	(* After writting, it is necessary to check if the parameter has been writting correctly*)
	Voltage_Guard_Min_Error_L1_RD(
		sNetId:= netID_internal,
		nSlaveAddr := Slave_Add_global_assign, 
		nIndex:= 16#8001, 
		nSubIndex := 16#11, 
		pDstBuf:= ADR(Voltage_Guard_Min_Error_L1), 
		cbBufLen:=SIZEOF(Voltage_Guard_Min_Error_L1),
		bExecute:= Exec_READ_Voltage_Guard_Min_Error_L1);
	
	(* Logic to handle the errors in the reading*)	
	IF NOT Voltage_Guard_Min_Error_L1_RD.bBusy AND NOT Voltage_Guard_Min_Error_L1_WR.bBusy THEN
    	Exec_READ_Voltage_Guard_Min_Error_L1 := FALSE;
		IF NOT Voltage_Guard_Min_Error_L1_RD.bError THEN 
			(* write successful *)
			Error_Voltage_Guard_Min_Error_L1 := FALSE;
			Previous_Voltage_Guard_Min_Error_L1_val := Voltage_Guard_Min_Error_L1;
		ELSE 
			(* write failed *)
			Error_Voltage_Guard_Min_Error_L1 := Voltage_Guard_Min_Error_L1_RD.bError;
    END_IF

    Voltage_Guard_Min_Error_L1_RD(bExecute := FALSE);
	
	END_IF
(******************************** VOLTAGE GUARD MIN ERROR L1 *****************************************)

(********************************* VOLTAGE GUARD MIN ERROR L2 ****************************************)
	(* Execution of the writing reading of Voltage Guard Min Error L2. When the previous value is diferent to the
	current one, the is executed the command*)
	IF Voltage_Guard_Min_Error_L2 <> Previous_Voltage_Guard_Min_Error_L2_val THEN
		Exec_Voltage_Guard_Min_Error_L2 := TRUE;
	END_IF
	
	(* Function to write the new value in the CoE parameter*)
	Voltage_Guard_Min_Error_L2_WR(
		sNetId:= netID_internal, 
		nSlaveAddr:= Slave_Add_global_assign, 
		nSubIndex:= 16#11, 
		nIndex:= 16#8011, 
		pSrcBuf:= ADR(Voltage_Guard_Min_Error_L2), 
		cbBufLen:= SIZEOF(Voltage_Guard_Min_Error_L2), 
		bExecute:= Exec_Voltage_Guard_Min_Error_L2, 
		tTimeout:= T#1S);
	
	(* Logic to handle the errors and launch the reading*)	
	IF NOT Voltage_Guard_Min_Error_L2_WR.bBusy THEN
    	Exec_Voltage_Guard_Min_Error_L2 := FALSE;
		IF NOT Voltage_Guard_Min_Error_L2_WR.bError THEN 
			(* write successful *)
			Error_Voltage_Guard_Min_Error_L2 := FALSE;
			IF Previous_Voltage_Guard_Min_Error_L2_val <> Voltage_Guard_Min_Error_L2 THEN
				Previous_Voltage_Guard_Min_Error_L2_val := Voltage_Guard_Min_Error_L2;
				Exec_READ_Voltage_Guard_Min_Error_L2 := TRUE;
			END_IF
		ELSE 
			(* write failed *)
			Error_Voltage_Guard_Min_Error_L2 := Voltage_Guard_Min_Error_L2_WR.bError;
			Voltage_Guard_Min_Error_L2 := Previous_Voltage_Guard_Min_Error_L2_val;
		END_IF
	
		Voltage_Guard_Min_Error_L2_WR(bExecute := FALSE);
	
	END_IF
	
	(* After writting, it is necessary to check if the parameter has been writting correctly*)
	Voltage_Guard_Min_Error_L2_RD(
		sNetId:= netID_internal,
		nSlaveAddr := Slave_Add_global_assign, 
		nIndex:= 16#8011, 
		nSubIndex := 16#11, 
		pDstBuf:= ADR(Voltage_Guard_Min_Error_L2), 
		cbBufLen:=SIZEOF(Voltage_Guard_Min_Error_L2),
		bExecute:= Exec_READ_Voltage_Guard_Min_Error_L2);
	
	(* Logic to handle the errors in the reading*)	
	IF NOT Voltage_Guard_Min_Error_L2_RD.bBusy AND NOT Voltage_Guard_Min_Error_L2_WR.bBusy THEN
    	Exec_READ_Voltage_Guard_Min_Error_L2 := FALSE;
		IF NOT Voltage_Guard_Min_Error_L2_RD.bError THEN 
			(* write successful *)
			Error_Voltage_Guard_Min_Error_L2 := FALSE;
			Previous_Voltage_Guard_Min_Error_L2_val := Voltage_Guard_Min_Error_L2;
		ELSE 
			(* write failed *)
			Error_Voltage_Guard_Min_Error_L2 := Voltage_Guard_Min_Error_L2_RD.bError;
    END_IF

    Voltage_Guard_Min_Error_L2_RD(bExecute := FALSE);
	
	END_IF
(********************************* VOLTAGE GUARD MIN ERROR L2 ****************************************)

(********************************* VOLTAGE GUARD MIN ERROR L3 ****************************************)
	(* Execution of the writing reading of Voltage Guard Min Error L23. When the previous value is diferent to the
	current one, the is executed the command*)
	IF Voltage_Guard_Min_Error_L3 <> Previous_Voltage_Guard_Min_Error_L3_val THEN
		Exec_Voltage_Guard_Min_Error_L3 := TRUE;
	END_IF
	
	(* Function to write the new value in the CoE parameter*)
	Voltage_Guard_Min_Error_L3_WR(
		sNetId:= netID_internal, 
		nSlaveAddr:= Slave_Add_global_assign, 
		nSubIndex:= 16#11, 
		nIndex:= 16#8021, 
		pSrcBuf:= ADR(Voltage_Guard_Min_Error_L3), 
		cbBufLen:= SIZEOF(Voltage_Guard_Min_Error_L3), 
		bExecute:= Exec_Voltage_Guard_Min_Error_L3, 
		tTimeout:= T#1S);
	
	(* Logic to handle the errors and launch the reading*)	
	IF NOT Voltage_Guard_Min_Error_L3_WR.bBusy THEN
    	Exec_Voltage_Guard_Min_Error_L3 := FALSE;
		IF NOT Voltage_Guard_Min_Error_L3_WR.bError THEN 
			(* write successful *)
			Error_Voltage_Guard_Min_Error_L3 := FALSE;
			IF Previous_Voltage_Guard_Min_Error_L3_val <> Voltage_Guard_Min_Error_L3 THEN
				Previous_Voltage_Guard_Min_Error_L3_val := Voltage_Guard_Min_Error_L3;
				Exec_READ_Voltage_Guard_Min_Error_L3 := TRUE;
			END_IF
		ELSE 
			(* write failed *)
			Error_Voltage_Guard_Min_Error_L3 := Voltage_Guard_Min_Error_L3_WR.bError;
			Voltage_Guard_Min_Error_L3 := Previous_Voltage_Guard_Min_Error_L3_val;
		END_IF
	
		Voltage_Guard_Min_Error_L3_WR(bExecute := FALSE);
	
	END_IF
	
	(* After writting, it is necessary to check if the parameter has been writting correctly*)
	Voltage_Guard_Min_Error_L3_RD(
		sNetId:= netID_internal,
		nSlaveAddr := Slave_Add_global_assign, 
		nIndex:= 16#8021, 
		nSubIndex := 16#11, 
		pDstBuf:= ADR(Voltage_Guard_Min_Error_L3), 
		cbBufLen:=SIZEOF(Voltage_Guard_Min_Error_L3),
		bExecute:= Exec_READ_Voltage_Guard_Min_Error_L3);
	
	(* Logic to handle the errors in the reading*)	
	IF NOT Voltage_Guard_Min_Error_L3_RD.bBusy AND NOT Voltage_Guard_Min_Error_L3_WR.bBusy THEN
    	Exec_READ_Voltage_Guard_Min_Error_L3 := FALSE;
		IF NOT Voltage_Guard_Min_Error_L3_RD.bError THEN 
			(* write successful *)
			Error_Voltage_Guard_Min_Error_L3 := FALSE;
			Previous_Voltage_Guard_Min_Error_L3_val := Voltage_Guard_Min_Error_L3;
		ELSE 
			(* write failed *)
			Error_Voltage_Guard_Min_Error_L3 := Voltage_Guard_Min_Error_L3_RD.bError;
    END_IF

    Voltage_Guard_Min_Error_L3_RD(bExecute := FALSE);
	
	END_IF
(******************************** VOLTAGE GUARD MIN ERROR L3 *****************************************)

(********************************* VOLTAGE GUARD MIN WARNING L1 **************************************)
	(* Execution of the writing reading of Voltage Guard Min Error L1. When the previous value is diferent to the
	current one, the is executed the command*)
	IF Voltage_Guard_Min_Warning_L1 <> Previous_Voltage_Guard_Min_Warning_L1_val THEN
		Exec_Voltage_Guard_Min_Warning_L1 := TRUE;
	END_IF
	
	(* Function to write the new value in the CoE parameter*)
	Voltage_Guard_Min_Warning_L1_WR(
		sNetId:= netID_internal, 
		nSlaveAddr:= Slave_Add_global_assign, 
		nSubIndex:= 16#12, 
		nIndex:= 16#8001, 
		pSrcBuf:= ADR(Voltage_Guard_Min_Warning_L1), 
		cbBufLen:= SIZEOF(Voltage_Guard_Min_Warning_L1), 
		bExecute:= Exec_Voltage_Guard_Min_Warning_L1, 
		tTimeout:= T#1S);
	
	(* Logic to handle the errors and launch the reading*)	
	IF NOT Voltage_Guard_Min_Warning_L1_WR.bBusy THEN
    	Exec_Voltage_Guard_Min_Warning_L1 := FALSE;
		IF NOT Voltage_Guard_Min_Warning_L1_WR.bError THEN 
			(* write successful *)
			Error_Voltage_Guard_Min_Warning_L1 := FALSE;
			IF Previous_Voltage_Guard_Min_Warning_L1_val <> Voltage_Guard_Min_Warning_L1 THEN
				Previous_Voltage_Guard_Min_Warning_L1_val := Voltage_Guard_Min_Warning_L1;
				Exec_READ_Voltage_Guard_Min_Warning_L1 := TRUE;
			END_IF
		ELSE 
			(* write failed *)
			Error_Voltage_Guard_Min_Warning_L1 := Voltage_Guard_Min_Warning_L1_WR.bError;
			Voltage_Guard_Min_Warning_L1 := Previous_Voltage_Guard_Min_Warning_L1_val;
		END_IF
	
		Voltage_Guard_Min_Warning_L1_WR(bExecute := FALSE);
	
	END_IF
	
	(* After writting, it is necessary to check if the parameter has been writting correctly*)
	Voltage_Guard_Min_Warning_L1_RD(
		sNetId:= netID_internal,
		nSlaveAddr := Slave_Add_global_assign, 
		nIndex:= 16#8001, 
		nSubIndex := 16#12, 
		pDstBuf:= ADR(Voltage_Guard_Min_Warning_L1), 
		cbBufLen:=SIZEOF(Voltage_Guard_Min_Warning_L1),
		bExecute:= Exec_READ_Voltage_Guard_Min_Warning_L1);
	
	(* Logic to handle the errors in the reading*)	
	IF NOT Voltage_Guard_Min_Warning_L1_RD.bBusy AND NOT Voltage_Guard_Min_Warning_L1_WR.bBusy THEN
    	Exec_READ_Voltage_Guard_Min_Warning_L1 := FALSE;
		IF NOT Voltage_Guard_Min_Warning_L1_RD.bError THEN 
			(* write successful *)
			Error_Voltage_Guard_Min_Warning_L1 := FALSE;
			Previous_Voltage_Guard_Min_Warning_L1_val := Voltage_Guard_Min_Warning_L1;
		ELSE 
			(* write failed *)
			Error_Voltage_Guard_Min_Warning_L1 := Voltage_Guard_Min_Warning_L1_RD.bError;
    END_IF

    Voltage_Guard_Min_Warning_L1_RD(bExecute := FALSE);
	
	END_IF
(********************************* VOLTAGE GUARD MIN WARNING L1 **************************************)

(********************************* VOLTAGE GUARD MIN WARNING L2 **************************************)
	(* Execution of the writing reading of Voltage Guard Min Error L2. When the previous value is diferent to the
	current one, the is executed the command*)
	IF Voltage_Guard_Min_Warning_L2 <> Previous_Voltage_Guard_Min_Warning_L2_val THEN
		Exec_Voltage_Guard_Min_Warning_L2 := TRUE;
	END_IF
	
	(* Function to write the new value in the CoE parameter*)
	Voltage_Guard_Min_Warning_L2_WR(
		sNetId:= netID_internal, 
		nSlaveAddr:= Slave_Add_global_assign, 
		nSubIndex:= 16#12, 
		nIndex:= 16#8011, 
		pSrcBuf:= ADR(Voltage_Guard_Min_Warning_L2), 
		cbBufLen:= SIZEOF(Voltage_Guard_Min_Warning_L2), 
		bExecute:= Exec_Voltage_Guard_Min_Warning_L2, 
		tTimeout:= T#1S);
	
	(* Logic to handle the errors and launch the reading*)	
	IF NOT Voltage_Guard_Min_Warning_L2_WR.bBusy THEN
    	Exec_Voltage_Guard_Min_Warning_L2 := FALSE;
		IF NOT Voltage_Guard_Min_Warning_L2_WR.bError THEN 
			(* write successful *)
			Error_Voltage_Guard_Min_Warning_L2 := FALSE;
			IF Previous_Voltage_Guard_Min_Warning_L2_val <> Voltage_Guard_Min_Warning_L2 THEN
				Previous_Voltage_Guard_Min_Warning_L2_val := Voltage_Guard_Min_Warning_L2;
				Exec_READ_Voltage_Guard_Min_Warning_L2 := TRUE;
			END_IF
		ELSE 
			(* write failed *)
			Error_Voltage_Guard_Min_Warning_L2 := Voltage_Guard_Min_Warning_L2_WR.bError;
			Voltage_Guard_Min_Warning_L2 := Previous_Voltage_Guard_Min_Warning_L2_val;
		END_IF
	
		Voltage_Guard_Min_Warning_L2_WR(bExecute := FALSE);
	
	END_IF
	
	(* After writting, it is necessary to check if the parameter has been writting correctly*)
	Voltage_Guard_Min_Warning_L2_RD(
		sNetId:= netID_internal,
		nSlaveAddr := Slave_Add_global_assign, 
		nIndex:= 16#8011, 
		nSubIndex := 16#12, 
		pDstBuf:= ADR(Voltage_Guard_Min_Warning_L2), 
		cbBufLen:=SIZEOF(Voltage_Guard_Min_Warning_L2),
		bExecute:= Exec_READ_Voltage_Guard_Min_Warning_L2);
	
	(* Logic to handle the errors in the reading*)	
	IF NOT Voltage_Guard_Min_Warning_L2_RD.bBusy AND NOT Voltage_Guard_Min_Warning_L2_WR.bBusy THEN
    	Exec_READ_Voltage_Guard_Min_Warning_L2 := FALSE;
		IF NOT Voltage_Guard_Min_Warning_L2_RD.bError THEN 
			(* write successful *)
			Error_Voltage_Guard_Min_Warning_L2 := FALSE;
			Previous_Voltage_Guard_Min_Warning_L2_val := Voltage_Guard_Min_Warning_L2;
		ELSE 
			(* write failed *)
			Error_Voltage_Guard_Min_Warning_L2 := Voltage_Guard_Min_Warning_L2_RD.bError;
    END_IF

    Voltage_Guard_Min_Warning_L2_RD(bExecute := FALSE);
	
	END_IF
(********************************* VOLTAGE GUARD MIN WARNING L2 ***************************************)

(********************************* VOLTAGE GUARD MIN WARNING L3 **************************************)
	(* Execution of the writing reading of Voltage Guard Min Error L3. When the previous value is diferent to the
	current one, the is executed the command*)
	IF Voltage_Guard_Min_Warning_L3 <> Previous_Voltage_Guard_Min_Warning_L3_val THEN
		Exec_Voltage_Guard_Min_Warning_L3 := TRUE;
	END_IF
	
	(* Function to write the new value in the CoE parameter*)
	Voltage_Guard_Min_Warning_L3_WR(
		sNetId:= netID_internal, 
		nSlaveAddr:= Slave_Add_global_assign, 
		nSubIndex:= 16#12, 
		nIndex:= 16#8021, 
		pSrcBuf:= ADR(Voltage_Guard_Min_Warning_L3), 
		cbBufLen:= SIZEOF(Voltage_Guard_Min_Warning_L3), 
		bExecute:= Exec_Voltage_Guard_Min_Warning_L3, 
		tTimeout:= T#1S);
	
	(* Logic to handle the errors and launch the reading*)	
	IF NOT Voltage_Guard_Min_Warning_L3_WR.bBusy THEN
    	Exec_Voltage_Guard_Min_Warning_L3 := FALSE;
		IF NOT Voltage_Guard_Min_Warning_L3_WR.bError THEN 
			(* write successful *)
			Error_Voltage_Guard_Min_Warning_L3 := FALSE;
			IF Previous_Voltage_Guard_Min_Warning_L3_val <> Voltage_Guard_Min_Warning_L3 THEN
				Previous_Voltage_Guard_Min_Warning_L3_val := Voltage_Guard_Min_Warning_L3;
				Exec_READ_Voltage_Guard_Min_Warning_L3 := TRUE;
			END_IF
		ELSE 
			(* write failed *)
			Error_Voltage_Guard_Min_Warning_L3 := Voltage_Guard_Min_Warning_L3_WR.bError;
			Voltage_Guard_Min_Warning_L3 := Previous_Voltage_Guard_Min_Warning_L3_val;
		END_IF
	
		Voltage_Guard_Min_Warning_L3_WR(bExecute := FALSE);
	
	END_IF
	
	(* After writting, it is necessary to check if the parameter has been writting correctly*)
	Voltage_Guard_Min_Warning_L3_RD(
		sNetId:= netID_internal,
		nSlaveAddr := Slave_Add_global_assign, 
		nIndex:= 16#8021, 
		nSubIndex := 16#12, 
		pDstBuf:= ADR(Voltage_Guard_Min_Warning_L3), 
		cbBufLen:=SIZEOF(Voltage_Guard_Min_Warning_L3),
		bExecute:= Exec_READ_Voltage_Guard_Min_Warning_L3);
	
	(* Logic to handle the errors in the reading*)	
	IF NOT Voltage_Guard_Min_Warning_L3_RD.bBusy AND NOT Voltage_Guard_Min_Warning_L3_WR.bBusy THEN
    	Exec_READ_Voltage_Guard_Min_Warning_L3 := FALSE;
		IF NOT Voltage_Guard_Min_Warning_L3_RD.bError THEN 
			(* write successful *)
			Error_Voltage_Guard_Min_Warning_L3 := FALSE;
			Previous_Voltage_Guard_Min_Warning_L3_val := Voltage_Guard_Min_Warning_L3;
		ELSE 
			(* write failed *)
			Error_Voltage_Guard_Min_Warning_L3 := Voltage_Guard_Min_Warning_L3_RD.bError;
    END_IF

    Voltage_Guard_Min_Warning_L3_RD(bExecute := FALSE);
	
	END_IF
(********************************* VOLTAGE GUARD MIN WARNING L3 ***************************************)

(********************************* VOLTAGE GUARD MAX WARNING L1 **************************************)
	(* Execution of the writing reading of Voltage Guard Max Warning L1. When the previous value is diferent to the
	current one, the is executed the command*)
	IF Voltage_Guard_Max_Warning_L1 <> Previous_Voltage_Guard_Max_Warning_L1_val THEN
		Exec_Voltage_Guard_Max_Warning_L1 := TRUE;
	END_IF
	
	(* Function to write the new value in the CoE parameter*)
	Voltage_Guard_Max_Warning_L1_WR(
		sNetId:= netID_internal, 
		nSlaveAddr:= Slave_Add_global_assign, 
		nSubIndex:= 16#13, 
		nIndex:= 16#8001, 
		pSrcBuf:= ADR(Voltage_Guard_Max_Warning_L1), 
		cbBufLen:= SIZEOF(Voltage_Guard_Max_Warning_L1), 
		bExecute:= Exec_Voltage_Guard_Max_Warning_L1, 
		tTimeout:= T#1S);
	
	(* Logic to handle the errors and launch the reading*)	
	IF NOT Voltage_Guard_Max_Warning_L1_WR.bBusy THEN
    	Exec_Voltage_Guard_Max_Warning_L1 := FALSE;
		IF NOT Voltage_Guard_Max_Warning_L1_WR.bError THEN 
			(* write successful *)
			Error_Voltage_Guard_Max_Warning_L1 := FALSE;
			IF Previous_Voltage_Guard_Max_Warning_L1_val <> Voltage_Guard_Max_Warning_L1 THEN
				Previous_Voltage_Guard_Max_Warning_L1_val := Voltage_Guard_Max_Warning_L1;
				Exec_READ_Voltage_Guard_Max_Warning_L1 := TRUE;
			END_IF
		ELSE 
			(* write failed *)
			Error_Voltage_Guard_Max_Warning_L1 := Voltage_Guard_Max_Warning_L1_WR.bError;
			Voltage_Guard_Max_Warning_L1 := Previous_Voltage_Guard_Max_Warning_L1_val;
		END_IF
	
		Voltage_Guard_Max_Warning_L1_WR(bExecute := FALSE);
	
	END_IF
	
	(* After writting, it is necessary to check if the parameter has been writting correctly*)
	Voltage_Guard_Max_Warning_L1_RD(
		sNetId:= netID_internal,
		nSlaveAddr := Slave_Add_global_assign, 
		nIndex:= 16#8001, 
		nSubIndex := 16#13, 
		pDstBuf:= ADR(Voltage_Guard_Max_Warning_L1), 
		cbBufLen:=SIZEOF(Voltage_Guard_Max_Warning_L1),
		bExecute:= Exec_READ_Voltage_Guard_Max_Warning_L1);
	
	(* Logic to handle the errors in the reading*)	
	IF NOT Voltage_Guard_Max_Warning_L1_RD.bBusy AND NOT Voltage_Guard_Max_Warning_L1_WR.bBusy THEN
    	Exec_READ_Voltage_Guard_Max_Warning_L1 := FALSE;
		IF NOT Voltage_Guard_Max_Warning_L1_RD.bError THEN 
			(* write successful *)
			Error_Voltage_Guard_Max_Warning_L1 := FALSE;
			Previous_Voltage_Guard_Max_Warning_L1_val := Voltage_Guard_Max_Warning_L1;
		ELSE 
			(* write failed *)
			Error_Voltage_Guard_Max_Warning_L1 := Voltage_Guard_Max_Warning_L1_RD.bError;
    END_IF

    Voltage_Guard_Max_Warning_L1_RD(bExecute := FALSE);
	
	END_IF
(********************************* VOLTAGE GUARD MAX WARNING L1 **************************************)

(********************************* VOLTAGE GUARD MAX WARNING L2 **************************************)
	(* Execution of the writing reading of Voltage Guard Max Warning L2. When the previous value is diferent to the
	current one, the is executed the command*)
	IF Voltage_Guard_Max_Warning_L2 <> Previous_Voltage_Guard_Max_Warning_L2_val THEN
		Exec_Voltage_Guard_Max_Warning_L2 := TRUE;
	END_IF
	
	(* Function to write the new value in the CoE parameter*)
	Voltage_Guard_Max_Warning_L2_WR(
		sNetId:= netID_internal, 
		nSlaveAddr:= Slave_Add_global_assign, 
		nSubIndex:= 16#13, 
		nIndex:= 16#8011, 
		pSrcBuf:= ADR(Voltage_Guard_Max_Warning_L2), 
		cbBufLen:= SIZEOF(Voltage_Guard_Max_Warning_L2), 
		bExecute:= Exec_Voltage_Guard_Max_Warning_L2, 
		tTimeout:= T#1S);
	
	(* Logic to handle the errors and launch the reading*)	
	IF NOT Voltage_Guard_Max_Warning_L2_WR.bBusy THEN
    	Exec_Voltage_Guard_Max_Warning_L2 := FALSE;
		IF NOT Voltage_Guard_Max_Warning_L2_WR.bError THEN 
			(* write successful *)
			Error_Voltage_Guard_Max_Warning_L2 := FALSE;
			IF Previous_Voltage_Guard_Max_Warning_L2_val <> Voltage_Guard_Max_Warning_L2 THEN
				Previous_Voltage_Guard_Max_Warning_L2_val := Voltage_Guard_Max_Warning_L2;
				Exec_READ_Voltage_Guard_Max_Warning_L2 := TRUE;
			END_IF
		ELSE 
			(* write failed *)
			Error_Voltage_Guard_Max_Warning_L2 := Voltage_Guard_Max_Warning_L2_WR.bError;
			Voltage_Guard_Max_Warning_L2 := Previous_Voltage_Guard_Max_Warning_L2_val;
		END_IF
	
		Voltage_Guard_Max_Warning_L2_WR(bExecute := FALSE);
	
	END_IF
	
	(* After writting, it is necessary to check if the parameter has been writting correctly*)
	Voltage_Guard_Max_Warning_L2_RD(
		sNetId:= netID_internal,
		nSlaveAddr := Slave_Add_global_assign, 
		nIndex:= 16#8011, 
		nSubIndex := 16#13, 
		pDstBuf:= ADR(Voltage_Guard_Max_Warning_L2), 
		cbBufLen:=SIZEOF(Voltage_Guard_Max_Warning_L2),
		bExecute:= Exec_READ_Voltage_Guard_Max_Warning_L2);
	
	(* Logic to handle the errors in the reading*)	
	IF NOT Voltage_Guard_Max_Warning_L2_RD.bBusy AND NOT Voltage_Guard_Max_Warning_L2_WR.bBusy THEN
    	Exec_READ_Voltage_Guard_Max_Warning_L2 := FALSE;
		IF NOT Voltage_Guard_Max_Warning_L2_RD.bError THEN 
			(* write successful *)
			Error_Voltage_Guard_Max_Warning_L2 := FALSE;
			Previous_Voltage_Guard_Max_Warning_L2_val := Voltage_Guard_Max_Warning_L2;
		ELSE 
			(* write failed *)
			Error_Voltage_Guard_Max_Warning_L2 := Voltage_Guard_Max_Warning_L2_RD.bError;
    END_IF

    Voltage_Guard_Max_Warning_L2_RD(bExecute := FALSE);
	
	END_IF
(********************************* VOLTAGE GUARD MAX WARNING L2 **************************************)

(********************************* VOLTAGE GUARD MAX WARNING L3 **************************************)
	(* Execution of the writing reading of Voltage Guard Max Warning L3. When the previous value is diferent to the
	current one, the is executed the command*)
	IF Voltage_Guard_Max_Warning_L3 <> Previous_Voltage_Guard_Max_Warning_L3_val THEN
		Exec_Voltage_Guard_Max_Warning_L3 := TRUE;
	END_IF
	
	(* Function to write the new value in the CoE parameter*)
	Voltage_Guard_Max_Warning_L3_WR(
		sNetId:= netID_internal, 
		nSlaveAddr:= Slave_Add_global_assign, 
		nSubIndex:= 16#13, 
		nIndex:= 16#8021, 
		pSrcBuf:= ADR(Voltage_Guard_Max_Warning_L3), 
		cbBufLen:= SIZEOF(Voltage_Guard_Max_Warning_L3), 
		bExecute:= Exec_Voltage_Guard_Max_Warning_L3, 
		tTimeout:= T#1S);
	
	(* Logic to handle the errors and launch the reading*)	
	IF NOT Voltage_Guard_Max_Warning_L3_WR.bBusy THEN
    	Exec_Voltage_Guard_Max_Warning_L3 := FALSE;
		IF NOT Voltage_Guard_Max_Warning_L3_WR.bError THEN 
			(* write successful *)
			Error_Voltage_Guard_Max_Warning_L3 := FALSE;
			IF Previous_Voltage_Guard_Max_Warning_L3_val <> Voltage_Guard_Max_Warning_L3 THEN
				Previous_Voltage_Guard_Max_Warning_L3_val := Voltage_Guard_Max_Warning_L3;
				Exec_READ_Voltage_Guard_Max_Warning_L3 := TRUE;
			END_IF
		ELSE 
			(* write failed *)
			Error_Voltage_Guard_Max_Warning_L3 := Voltage_Guard_Max_Warning_L3_WR.bError;
			Voltage_Guard_Max_Warning_L3 := Previous_Voltage_Guard_Max_Warning_L3_val;
		END_IF
	
		Voltage_Guard_Max_Warning_L3_WR(bExecute := FALSE);
	
	END_IF
	
	(* After writting, it is necessary to check if the parameter has been writting correctly*)
	Voltage_Guard_Max_Warning_L3_RD(
		sNetId:= netID_internal,
		nSlaveAddr := Slave_Add_global_assign, 
		nIndex:= 16#8021, 
		nSubIndex := 16#13, 
		pDstBuf:= ADR(Voltage_Guard_Max_Warning_L3), 
		cbBufLen:=SIZEOF(Voltage_Guard_Max_Warning_L3),
		bExecute:= Exec_READ_Voltage_Guard_Max_Warning_L3);
	
	(* Logic to handle the errors in the reading*)	
	IF NOT Voltage_Guard_Max_Warning_L3_RD.bBusy AND NOT Voltage_Guard_Max_Warning_L3_WR.bBusy THEN
    	Exec_READ_Voltage_Guard_Max_Warning_L3 := FALSE;
		IF NOT Voltage_Guard_Max_Warning_L3_RD.bError THEN 
			(* write successful *)
			Error_Voltage_Guard_Max_Warning_L3 := FALSE;
			Previous_Voltage_Guard_Max_Warning_L3_val := Voltage_Guard_Max_Warning_L3;
		ELSE 
			(* write failed *)
			Error_Voltage_Guard_Max_Warning_L3 := Voltage_Guard_Max_Warning_L3_RD.bError;
    END_IF

    Voltage_Guard_Max_Warning_L3_RD(bExecute := FALSE);
	
	END_IF
(********************************* VOLTAGE GUARD MAX WARNING L3 **************************************)

(********************************* VOLTAGE GUARD MAX ERROR L1 ****************************************)
	(* Execution of the writing reading of Voltage Guard Max Error L1. When the previous value is diferent to the
	current one, the is executed the command*)
	IF Voltage_Guard_Max_Error_L1 <> Previous_Voltage_Guard_Max_Error_L1_val THEN
		Exec_Voltage_Guard_Max_Error_L1 := TRUE;
	END_IF
	
	(* Function to write the new value in the CoE parameter*)
	Voltage_Guard_Max_Error_L1_WR(
		sNetId:= netID_internal, 
		nSlaveAddr:= Slave_Add_global_assign, 
		nSubIndex:= 16#14, 
		nIndex:= 16#8001, 
		pSrcBuf:= ADR(Voltage_Guard_Max_Error_L1), 
		cbBufLen:= SIZEOF(Voltage_Guard_Max_Error_L1), 
		bExecute:= Exec_Voltage_Guard_Max_Error_L1, 
		tTimeout:= T#1S);
	
	(* Logic to handle the errors and launch the reading*)	
	IF NOT Voltage_Guard_Max_Error_L1_WR.bBusy THEN
    	Exec_Voltage_Guard_Max_Error_L1 := FALSE;
		IF NOT Voltage_Guard_Max_Error_L1_WR.bError THEN 
			(* write successful *)
			Error_Voltage_Guard_Max_Error_L1 := FALSE;
			IF Previous_Voltage_Guard_Max_Error_L1_val <> Voltage_Guard_Max_Error_L1 THEN
				Previous_Voltage_Guard_Max_Error_L1_val := Voltage_Guard_Max_Error_L1;
				Exec_READ_Voltage_Guard_Max_Error_L1 := TRUE;
			END_IF
		ELSE 
			(* write failed *)
			Error_Voltage_Guard_Max_Error_L1 := Voltage_Guard_Max_Error_L1_WR.bError;
			Voltage_Guard_Max_Error_L1 := Previous_Voltage_Guard_Max_Error_L1_val;
		END_IF
	
		Voltage_Guard_Max_Error_L1_WR(bExecute := FALSE);
	
	END_IF
	
	(* After writting, it is necessary to check if the parameter has been writting correctly*)
	Voltage_Guard_Max_Error_L1_RD(
		sNetId:= netID_internal,
		nSlaveAddr := Slave_Add_global_assign, 
		nIndex:= 16#8001, 
		nSubIndex := 16#14, 
		pDstBuf:= ADR(Voltage_Guard_Max_Error_L1), 
		cbBufLen:=SIZEOF(Voltage_Guard_Max_Error_L1),
		bExecute:= Exec_READ_Voltage_Guard_Max_Error_L1);
	
	(* Logic to handle the errors in the reading*)	
	IF NOT Voltage_Guard_Max_Error_L1_RD.bBusy AND NOT Voltage_Guard_Max_Error_L1_WR.bBusy THEN
    	Exec_READ_Voltage_Guard_Max_Error_L1 := FALSE;
		IF NOT Voltage_Guard_Max_Error_L1_RD.bError THEN 
			(* write successful *)
			Error_Voltage_Guard_Max_Error_L1 := FALSE;
			Previous_Voltage_Guard_Max_Error_L1_val := Voltage_Guard_Max_Error_L1;
		ELSE 
			(* write failed *)
			Error_Voltage_Guard_Max_Error_L1 := Voltage_Guard_Max_Error_L1_RD.bError;
    END_IF

    Voltage_Guard_Max_Error_L1_RD(bExecute := FALSE);
	
	END_IF
(******************************** VOLTAGE GUARD MAX ERROR L1 *****************************************)

(********************************* VOLTAGE GUARD MAX ERROR L2 ****************************************)
	(* Execution of the writing reading of Voltage Guard Max Error L2. When the previous value is diferent to the
	current one, the is executed the command*)
	IF Voltage_Guard_Max_Error_L2 <> Previous_Voltage_Guard_Max_Error_L2_val THEN
		Exec_Voltage_Guard_Max_Error_L2 := TRUE;
	END_IF
	
	(* Function to write the new value in the CoE parameter*)
	Voltage_Guard_Max_Error_L2_WR(
		sNetId:= netID_internal, 
		nSlaveAddr:= Slave_Add_global_assign, 
		nSubIndex:= 16#14, 
		nIndex:= 16#8011, 
		pSrcBuf:= ADR(Voltage_Guard_Max_Error_L2), 
		cbBufLen:= SIZEOF(Voltage_Guard_Max_Error_L2), 
		bExecute:= Exec_Voltage_Guard_Max_Error_L2, 
		tTimeout:= T#1S);
	
	(* Logic to handle the errors and launch the reading*)	
	IF NOT Voltage_Guard_Max_Error_L2_WR.bBusy THEN
    	Exec_Voltage_Guard_Max_Error_L2 := FALSE;
		IF NOT Voltage_Guard_Max_Error_L2_WR.bError THEN 
			(* write successful *)
			Error_Voltage_Guard_Max_Error_L2 := FALSE;
			IF Previous_Voltage_Guard_Max_Error_L2_val <> Voltage_Guard_Max_Error_L2 THEN
				Previous_Voltage_Guard_Max_Error_L2_val := Voltage_Guard_Max_Error_L2;
				Exec_READ_Voltage_Guard_Max_Error_L2 := TRUE;
			END_IF
		ELSE 
			(* write failed *)
			Error_Voltage_Guard_Max_Error_L2 := Voltage_Guard_Max_Error_L2_WR.bError;
			Voltage_Guard_Max_Error_L2 := Previous_Voltage_Guard_Max_Error_L2_val;
		END_IF
	
		Voltage_Guard_Max_Error_L2_WR(bExecute := FALSE);
	
	END_IF
	
	(* After writting, it is necessary to check if the parameter has been writting correctly*)
	Voltage_Guard_Max_Error_L2_RD(
		sNetId:= netID_internal,
		nSlaveAddr := Slave_Add_global_assign, 
		nIndex:= 16#8011, 
		nSubIndex := 16#14, 
		pDstBuf:= ADR(Voltage_Guard_Max_Error_L2), 
		cbBufLen:=SIZEOF(Voltage_Guard_Max_Error_L2),
		bExecute:= Exec_READ_Voltage_Guard_Max_Error_L2);
	
	(* Logic to handle the errors in the reading*)	
	IF NOT Voltage_Guard_Max_Error_L2_RD.bBusy AND NOT Voltage_Guard_Max_Error_L2_WR.bBusy THEN
    	Exec_READ_Voltage_Guard_Max_Error_L2 := FALSE;
		IF NOT Voltage_Guard_Max_Error_L2_RD.bError THEN 
			(* write successful *)
			Error_Voltage_Guard_Max_Error_L2 := FALSE;
			Previous_Voltage_Guard_Max_Error_L2_val := Voltage_Guard_Max_Error_L2;
		ELSE 
			(* write failed *)
			Error_Voltage_Guard_Max_Error_L2 := Voltage_Guard_Max_Error_L2_RD.bError;
    END_IF

    Voltage_Guard_Max_Error_L2_RD(bExecute := FALSE);
	
	END_IF
(******************************** VOLTAGE GUARD MAX ERROR L2 *****************************************)

(********************************* VOLTAGE GUARD MAX ERROR L3 ****************************************)
	(* Execution of the writing reading of Voltage Guard Max Error L3. When the previous value is diferent to the
	current one, the is executed the command*)
	IF Voltage_Guard_Max_Error_L3 <> Previous_Voltage_Guard_Max_Error_L3_val THEN
		Exec_Voltage_Guard_Max_Error_L3 := TRUE;
	END_IF
	
	(* Function to write the new value in the CoE parameter*)
	Voltage_Guard_Max_Error_L3_WR(
		sNetId:= netID_internal, 
		nSlaveAddr:= Slave_Add_global_assign, 
		nSubIndex:= 16#14, 
		nIndex:= 16#8021, 
		pSrcBuf:= ADR(Voltage_Guard_Max_Error_L3), 
		cbBufLen:= SIZEOF(Voltage_Guard_Max_Error_L3), 
		bExecute:= Exec_Voltage_Guard_Max_Error_L3, 
		tTimeout:= T#1S);
	
	(* Logic to handle the errors and launch the reading*)	
	IF NOT Voltage_Guard_Max_Error_L3_WR.bBusy THEN
    	Exec_Voltage_Guard_Max_Error_L3 := FALSE;
		IF NOT Voltage_Guard_Max_Error_L3_WR.bError THEN 
			(* write successful *)
			Error_Voltage_Guard_Max_Error_L3 := FALSE;
			IF Previous_Voltage_Guard_Max_Error_L3_val <> Voltage_Guard_Max_Error_L3 THEN
				Previous_Voltage_Guard_Max_Error_L3_val := Voltage_Guard_Max_Error_L3;
				Exec_READ_Voltage_Guard_Max_Error_L3 := TRUE;
			END_IF
		ELSE 
			(* write failed *)
			Error_Voltage_Guard_Max_Error_L3 := Voltage_Guard_Max_Error_L3_WR.bError;
			Voltage_Guard_Max_Error_L3 := Previous_Voltage_Guard_Max_Error_L3_val;
		END_IF
	
		Voltage_Guard_Max_Error_L3_WR(bExecute := FALSE);
	
	END_IF
	
	(* After writting, it is necessary to check if the parameter has been writting correctly*)
	Voltage_Guard_Max_Error_L3_RD(
		sNetId:= netID_internal,
		nSlaveAddr := Slave_Add_global_assign, 
		nIndex:= 16#8021, 
		nSubIndex := 16#14, 
		pDstBuf:= ADR(Voltage_Guard_Max_Error_L3), 
		cbBufLen:=SIZEOF(Voltage_Guard_Max_Error_L3),
		bExecute:= Exec_READ_Voltage_Guard_Max_Error_L3);
	
	(* Logic to handle the errors in the reading*)	
	IF NOT Voltage_Guard_Max_Error_L3_RD.bBusy AND NOT Voltage_Guard_Max_Error_L3_WR.bBusy THEN
    	Exec_READ_Voltage_Guard_Max_Error_L3 := FALSE;
		IF NOT Voltage_Guard_Max_Error_L3_RD.bError THEN 
			(* write successful *)
			Error_Voltage_Guard_Max_Error_L3 := FALSE;
			Previous_Voltage_Guard_Max_Error_L3_val := Voltage_Guard_Max_Error_L3;
		ELSE 
			(* write failed *)
			Error_Voltage_Guard_Max_Error_L3 := Voltage_Guard_Max_Error_L3_RD.bError;
    END_IF

    Voltage_Guard_Max_Error_L3_RD(bExecute := FALSE);
	
	END_IF
(******************************** VOLTAGE GUARD MAX ERROR L3 *****************************************)

END_IF

IF EL3_Selection = 'EL3453' THEN
	
	(* Reset the error selection *)
	Error_selection := FALSE;
	
	
(********************************** CURRENT TRAFO RANGE L1 *******************************************)
	(* Execution of the writing reading of nominal voltage. When the previous value is diferent to the
	current one, the is executed the command*)
	IF Current_trafo_range_L1 <> Previous_Current_trafo_range_L1_val THEN
		Exec_Current_trafo_range_L1 := TRUE;
	END_IF
	
	(* Function to write the new value in the CoE parameter*)
	Current_trafo_range_L1_WR(
		sNetId:= netID_internal, 
		nSlaveAddr:= Slave_Add_global_assign, 
		nSubIndex:= 16#14, 
		nIndex:= 16#8000, 
		pSrcBuf:= ADR(Current_trafo_range_L1), 
		cbBufLen:= SIZEOF(Current_trafo_range_L1), 
		bExecute:= Exec_Current_trafo_range_L1, 
		tTimeout:= T#1S);
	
	(* Logic to handle the errors and launch the reading*)	
	IF NOT Current_trafo_range_L1_WR.bBusy THEN
    	Exec_Current_trafo_range_L1 := FALSE;
		IF NOT Current_trafo_range_L1_WR.bError THEN 
			(* write successful *)
			Error_Current_trafo_range_L1 := FALSE;
			IF Previous_Current_trafo_range_L1_val <> Current_trafo_range_L1 THEN
				Previous_Current_trafo_range_L1_val := Current_trafo_range_L1;
				Exec_READ_Current_trafo_range_L1 := TRUE;
			END_IF
		ELSE 
			(* write failed *)
			Error_Current_trafo_range_L1 := Current_trafo_range_L1_WR.bError;
			Current_trafo_range_L1 := Previous_Current_trafo_range_L1_val;
		END_IF
	
		Current_trafo_range_L1_WR(bExecute := FALSE);
	
	END_IF
	
	(* After writting, it is necessary to check if the parameter has been writting correctly*)
	Current_trafo_range_L1_RD(
		sNetId:= netID_internal,
		nSlaveAddr := Slave_Add_global_assign, 
		nIndex:= 16#8000, 
		nSubIndex := 16#14, 
		pDstBuf:= ADR(Current_trafo_range_L1), 
		cbBufLen:=SIZEOF(Current_trafo_range_L1),
		bExecute:= Exec_READ_Current_trafo_range_L1);
	
	(* Logic to handle the errors in the reading*)	
	IF NOT Current_trafo_range_L1_RD.bBusy AND NOT Current_trafo_range_L1_WR.bBusy THEN
    	Exec_READ_Current_trafo_range_L1 := FALSE;
		IF NOT Current_trafo_range_L1_RD.bError THEN 
			(* write successful *)
			Error_Current_trafo_range_L1 := FALSE;
			Previous_Current_trafo_range_L1_val := Current_trafo_range_L1;
		ELSE 
			(* write failed *)
			Error_Current_trafo_range_L1 := Current_trafo_range_L1_RD.bError;
    	END_IF

    Current_trafo_range_L1_RD(bExecute := FALSE);
	
	END_IF
	
(********************************** CURRENT TRAFO RANGE L1 *******************************************)

(********************************** CURRENT TRAFO RANGE L2 *******************************************)
	(* Execution of the writing reading of nominal voltage. When the previous value is diferent to the
	current one, the is executed the command*)
	IF Current_trafo_range_L2 <> Previous_Current_trafo_range_L2_val THEN
		Exec_Current_trafo_range_L2 := TRUE;
	END_IF
	
	(* Function to write the new value in the CoE parameter*)
	Current_trafo_range_L2_WR(
		sNetId:= netID_internal, 
		nSlaveAddr:= Slave_Add_global_assign, 
		nSubIndex:= 16#14, 
		nIndex:= 16#8010, 
		pSrcBuf:= ADR(Current_trafo_range_L2), 
		cbBufLen:= SIZEOF(Current_trafo_range_L2), 
		bExecute:= Exec_Current_trafo_range_L2, 
		tTimeout:= T#1S);
	
	(* Logic to handle the errors and launch the reading*)	
	IF NOT Current_trafo_range_L2_WR.bBusy THEN
    	Exec_Current_trafo_range_L2 := FALSE;
		IF NOT Current_trafo_range_L2_WR.bError THEN 
			(* write successful *)
			Error_Current_trafo_range_L2 := FALSE;
			IF Previous_Current_trafo_range_L2_val <> Current_trafo_range_L2 THEN
				Previous_Current_trafo_range_L2_val := Current_trafo_range_L2;
				Exec_READ_Current_trafo_range_L2 := TRUE;
			END_IF
		ELSE 
			(* write failed *)
			Error_Current_trafo_range_L2 := Current_trafo_range_L2_WR.bError;
			Current_trafo_range_L2 := Previous_Current_trafo_range_L2_val;
		END_IF
	
		Current_trafo_range_L2_WR(bExecute := FALSE);
	
	END_IF
	
	(* After writting, it is necessary to check if the parameter has been writting correctly*)
	Current_trafo_range_L2_RD(
		sNetId:= netID_internal,
		nSlaveAddr := Slave_Add_global_assign, 
		nIndex:= 16#8010, 
		nSubIndex := 16#14, 
		pDstBuf:= ADR(Current_trafo_range_L2), 
		cbBufLen:=SIZEOF(Current_trafo_range_L2),
		bExecute:= Exec_READ_Current_trafo_range_L2);
	
	(* Logic to handle the errors in the reading*)	
	IF NOT Current_trafo_range_L2_RD.bBusy AND NOT Current_trafo_range_L2_WR.bBusy THEN
    	Exec_READ_Current_trafo_range_L2 := FALSE;
		IF NOT Current_trafo_range_L2_RD.bError THEN 
			(* write successful *)
			Error_Current_trafo_range_L2 := FALSE;
			Previous_Current_trafo_range_L2_val := Current_trafo_range_L2;
		ELSE 
			(* write failed *)
			Error_Current_trafo_range_L2 := Current_trafo_range_L2_RD.bError;
    	END_IF

    Current_trafo_range_L2_RD(bExecute := FALSE);
	
	END_IF
	
(********************************** CURRENT TRAFO RANGE L2 *******************************************)

(********************************** CURRENT TRAFO RANGE L3 *******************************************)
	(* Execution of the writing reading of nominal voltage. When the previous value is diferent to the
	current one, the is executed the command*)
	IF Current_trafo_range_L3 <> Previous_Current_trafo_range_L3_val THEN
		Exec_Current_trafo_range_L3 := TRUE;
	END_IF
	
	(* Function to write the new value in the CoE parameter*)
	Current_trafo_range_L3_WR(
		sNetId:= netID_internal, 
		nSlaveAddr:= Slave_Add_global_assign, 
		nSubIndex:= 16#14, 
		nIndex:= 16#8020, 
		pSrcBuf:= ADR(Current_trafo_range_L3), 
		cbBufLen:= SIZEOF(Current_trafo_range_L3), 
		bExecute:= Exec_Current_trafo_range_L3, 
		tTimeout:= T#1S);
	
	(* Logic to handle the errors and launch the reading*)	
	IF NOT Current_trafo_range_L3_WR.bBusy THEN
    	Exec_Current_trafo_range_L3 := FALSE;
		IF NOT Current_trafo_range_L3_WR.bError THEN 
			(* write successful *)
			Error_Current_trafo_range_L3 := FALSE;
			IF Previous_Current_trafo_range_L3_val <> Current_trafo_range_L3 THEN
				Previous_Current_trafo_range_L3_val := Current_trafo_range_L3;
				Exec_READ_Current_trafo_range_L3 := TRUE;
			END_IF
		ELSE 
			(* write failed *)
			Error_Current_trafo_range_L3 := Current_trafo_range_L3_WR.bError;
			Current_trafo_range_L3 := Previous_Current_trafo_range_L3_val;
		END_IF
	
		Current_trafo_range_L3_WR(bExecute := FALSE);
	
	END_IF
	
	(* After writting, it is necessary to check if the parameter has been writting correctly*)
	Current_trafo_range_L3_RD(
		sNetId:= netID_internal,
		nSlaveAddr := Slave_Add_global_assign, 
		nIndex:= 16#8020, 
		nSubIndex := 16#14, 
		pDstBuf:= ADR(Current_trafo_range_L3), 
		cbBufLen:=SIZEOF(Current_trafo_range_L3),
		bExecute:= Exec_READ_Current_trafo_range_L3);
	
	(* Logic to handle the errors in the reading*)	
	IF NOT Current_trafo_range_L3_RD.bBusy AND NOT Current_trafo_range_L3_WR.bBusy THEN
    	Exec_READ_Current_trafo_range_L3 := FALSE;
		IF NOT Current_trafo_range_L3_RD.bError THEN 
			(* write successful *)
			Error_Current_trafo_range_L3 := FALSE;
			Previous_Current_trafo_range_L3_val := Current_trafo_range_L3;
		ELSE 
			(* write failed *)
			Error_Current_trafo_range_L3 := Current_trafo_range_L3_RD.bError;
    	END_IF

    Current_trafo_range_L3_RD(bExecute := FALSE);
	
	END_IF
	
(********************************** CURRENT TRAFO RANGE L3 *******************************************)


END_IF

(* It is necessary to know what is the power measurement boards that is going to be configured *)	
IF EL3_Selection = 'EL3783' THEN
	
	(* In the first scan cycle, the function performs a reading to get the parameters from the board *)
	(* It is necessary send the request in two times, otherwise the last frames reports error*)
	
	IF INIT_THIRD = TRUE THEN	
		IF INIT AND Counter_Init_2 <= 1 THEN
			CASE Counter_init_2 OF
				//Current Range
				0: Exec_READ_Current_Range := TRUE;
				
			END_CASE
			Counter_init_2 := Counter_init_2 + 1;
		END_IF
	END_IF

	Delay_third_Init (IN := NOT(INIT_THIRD), PT := T#200MS, Q => INIT_THIRD, ET => );
	
	(* Reset the error selection *)
	Error_selection := FALSE;
	
(************************************** CURRENT RANGE **********************************************)
	(* Execution of the writing reading of Current Range. When the previous value is diferent to the
	current one, the is executed the command*)
	IF Current_Range <> Previous_Current_Range_val THEN
		Exec_Current_Range := TRUE;
	END_IF
	
	(* Function to write the new value in the CoE parameter*)
	Current_Range_WR(
		sNetId:= netID_internal_2, 
		nSlaveAddr:= Slave_Add_global_assign_2, 
		nSubIndex:= 16#11, 
		nIndex:= 16#F80D, 
		pSrcBuf:= ADR(Current_Range), 
		cbBufLen:= SIZEOF(Current_Range), 
		bExecute:= Exec_Current_Range, 
		tTimeout:= T#1S);
	
	(* Logic to handle the errors and launch the reading*)	
	IF NOT Current_Range_WR.bBusy THEN
    	Exec_Current_Range := FALSE;
		IF NOT Current_Range_WR.bError THEN 
			(* write successful *)
			Error_Current_Range := FALSE;
			IF Previous_Current_Range_val <> Current_Range THEN
				Previous_Current_Range_val := Current_Range;
				Exec_READ_Current_Range := TRUE;
			END_IF
		ELSE 
			(* write failed *)
			Error_Current_Range := Current_Range_WR.bError;
			Current_Range := Previous_Current_Range_val;
		END_IF
	
		Current_Range_WR(bExecute := FALSE);
	
	END_IF
	
	(* After writting, it is necessary to check if the parameter has been writting correctly*)
	Current_Range_RD(
		sNetId:= netID_internal_2,
		nSlaveAddr := Slave_Add_global_assign_2, 
		nIndex:= 16#F80D, 
		nSubIndex := 16#11, 
		pDstBuf:= ADR(Current_Range), 
		cbBufLen:=SIZEOF(Current_Range),
		bExecute:= Exec_READ_Current_Range);
	
	(* Logic to handle the errors in the reading*)	
	IF NOT Current_Range_RD.bBusy AND NOT Current_Range_WR.bBusy THEN
    	Exec_READ_Current_Range := FALSE;
		IF NOT Current_Range_RD.bError THEN 
			(* write successful *)
			Error_Current_Range := FALSE;
			Previous_Current_Range_val := Current_Range;
		ELSE 
			(* write failed *)
			Error_Current_Range := Current_Range_RD.bError;
    	END_IF

    	Current_Range_RD(bExecute := FALSE);
	
	END_IF
	
(********************************** CURRENT RANGE *******************************************)

END_IF

//If non of EL3443 or EL3453 or EL3783 is selected then "Error selection" became True
	
IF EL3_Selection <> 'EL3783' AND EL3_Selection <> 'EL3443' AND EL3_Selection <> 'EL3453' THEN 
	Error_selection := TRUE;
END_IF

END_FUNCTION_BLOCK

// ---- POUs/MAIN.TcPOU
PROGRAM MAIN
VAR
END_VAR

CONVERTERS_COMMS();

Parameters_handler();

END_PROGRAM

// ---- POUs/CONVERTERS/CONVERTERS_COMMS.TcPOU
PROGRAM CONVERTERS_COMMS
VAR
	I: word;//loop  variable
END_VAR

(*
 ************************************************************************************************************
 * \file  CONVERTERS_COMMS
 * \author Quique
 * \version 1.0.0
 * \date Creation: 15/06/2022
 * \date Modification: 12/08/2022
 * \brief Programm to handle / arrange communications with converters
 ************************************************************************************************************
 \defgroup CONVERTERS
 
 \brief 	This program takes P and Q from all algorithms to write it to all converters
		
 \details 	First part takes P and Q from algorithms and write them to converters
 			
 			Second part handles communications with metering board to accomplish I.3.4 from RD 244/19
			
			Third part writes relevant bits to inverters using a single modbus register, but bitwisely,
			so that
			
			bit 0 --> Stop / start command
			bit 1 --> Heartbeat to converters.
			bit 2 --> Night mode enabling.
 
*)

FOR I := 1 TO GVL_CONV_COMMS.NUMBER_CONVERTERS DO;
	
	GVL_CONV_COMMS.Setpoint_P[I] := REAL_TO_WORD(GVL_P_CONTROL.P_output);
	GVL_CONV_COMMS.Setpoint_Q[I] := REAL_TO_INT(GVL_Q_CONTROL.Q_output);

	//Powermeter loss comms section
	IF GVL_POWERMETER.Alg_lost_comms_enable THEN		
		IF GVL_POWERMETER.M_board_Meter_status <> 8 THEN
			GVL_CONV_COMMS.Setpoint_P[I] := REAL_TO_WORD(GVL_P_CONTROL.P_safety);
			GVL_CONV_COMMS.Setpoint_Q[I] := REAL_TO_INT(GVL_Q_CONTROL.Q_safety);
		END_IF
	END_IF
	
	CASE GVL_POWERMETER.M_board_Meter_status OF
		8: GVL_POWERMETER.Meter_comms_status:= TRUE;
		ELSE
			GVL_POWERMETER.Meter_comms_status:= FALSE;
	END_CASE
	
	IF ((GVL_CONV_COMMS.Comms_Control_Word[I] AND 16#0001) > 0 ) THEN
			GVL_CONV_COMMS.Start_Command[I] := 1;
		ELSE
			GVL_CONV_COMMS.Start_Command[I] := 0;
		END_IF
		
		IF ((GVL_CONV_COMMS.Comms_Control_Word[I] AND 16#0002) > 0 ) THEN
			GVL_CONV_COMMS.Night_Mode_Active[I] := 1;
		ELSE
			GVL_CONV_COMMS.Night_Mode_Active[I] := 0;
		END_IF
END_FOR;

//****************************************************************************************
//                               n/N COEFFICIENT
//****************************************************************************************

nN_coeff_calculation();

//****************************************************************************************
//                               MODBUS COMMS MAPPING
//****************************************************************************************

Modbus_mapping();

END_PROGRAM

// ---- POUs/CONVERTERS/nN_coeff_calculation.TcPOU
PROGRAM nN_coeff_calculation
VAR
	I: WORD;//loop  variable
	
	power_accumulated_run: REAL := 0;// Auxiliar accumulator
	
END_VAR

(*
***************************************************************************************************
* \file    nN coefficient calculation
* \author  Quique
* \version V1.0.0
* \date    12/08/2022
* \brief   Calculation of n/N coefficient
***************************************************************************************************

\brief   Code block used to calculate n/N coefficient for converters running

\details	This code looks which inverters are online and running (on state), understanding
			that those inverters are controllable by PPC. Then it takes the power of those
			controlable ones, sums it and compares with plant nominal power to obtain a 
			coefficient of the inverters' powers running and able to control with respect to 
			plant total.  
	     
*)

FOR I := 1 TO GVL_CONV_COMMS.NUMBER_CONVERTERS DO;
	
	IF GVL_CONV_COMMS.Current_Status[I] = GVL_CONVERTERS_COMMON.CONVERTER_STATUS_RUN AND GVL_CONV_COMMS.ERROR_TASK[I] <> 1 THEN
		//Only inverters in ON status and online are taken into account
		power_accumulated_run := power_accumulated_run + GVL_CONV_COMMS.CONVERTERS[I].Capacity;
	END_IF
END_FOR

GVL_CONV_COMMS.converters_nN_coeff := power_accumulated_run / GVL_PLANT_DEF.Plant_capacity_nom;
power_accumulated_run := 0;

END_PROGRAM

// ---- POUs/CONVERTERS/Modbus_mapping.TcPOU
PROGRAM Modbus_mapping
VAR
	I: WORD;//loop  variable

END_VAR



FOR I:=1 TO GVL_CONV_COMMS.NUMBER_CONVERTERS DO;
	//Reading Mapping
	GVL_CONV_COMMS.P_Measured[I] := GVL_CONV_COMMS.CONVERTERS[I].READING[1];
	GVL_CONV_COMMS.Q_Measured[I] := GVL_CONV_COMMS.CONVERTERS[I].READING[2];
	GVL_CONV_COMMS.S_Measured[I] := GVL_CONV_COMMS.CONVERTERS[I].READING[3];	
	GVL_CONV_COMMS.cosphi_Measured[I] := GVL_CONV_COMMS.CONVERTERS[I].READING[4];
	GVL_CONV_COMMS.Current_Status[I] := GVL_CONV_COMMS.CONVERTERS[I].READING[5];
	
	//Writting Mapping
	GVL_CONV_COMMS.CONVERTERS[I].WRITING[1]:= INT_TO_WORD(GVL_CONV_COMMS.Setpoint_Q [I]);
	GVL_CONV_COMMS.CONVERTERS[I].WRITING[2]:= GVL_CONV_COMMS.Setpoint_P [I];
	
	//GVL_CONV_COMMS.CONVERTERS[I].WRITING[3]:= INT_TO_WORD (GVL_CONV_COMMS.Start_Command[I]);
	//GVL_CONV_COMMS.CONVERTERS[I].WRITING[4]:= GVL_CONV_COMMS.Watchdog_PPC;
	//GVL_CONV_COMMS.CONVERTERS[I].WRITING[5]:= INT_TO_WORD (GVL_CONV_COMMS.Night_Mode_Active[I]);
	GVL_CONV_COMMS.CONVERTERS[I].WRITING[3]:= BIT_TO_WORD (GVL_CONV_COMMS.Comms_Control_Word[I].0);
	GVL_CONV_COMMS.CONVERTERS[I].WRITING[4]:= BIT_TO_WORD (GVL_CONV_COMMS.Comms_Control_Word[I].1);
	GVL_CONV_COMMS.CONVERTERS[I].WRITING[5]:= BIT_TO_WORD (GVL_CONV_COMMS.Comms_Control_Word[I].2);	
	
	GVL_CONV_COMMS.Status_Byte[I]:= WORD_TO_BYTE(GVL_CONV_COMMS.Current_Status[I]);
	GVL_CONV_COMMS.Control_Byte[I]:= WORD_TO_BYTE(GVL_CONV_COMMS.Comms_Control_Word[I]);
	
	GVL_CONV_COMMS.Comms_Control_Word[I]:= SHL(GVL_CONV_COMMS.Status_Byte[I], 7) + GVL_CONV_COMMS.Control_Byte[I];
END_FOR

END_PROGRAM

// ---- POUs/HANDLER_PARAM/Parameters_handler.TcPOU
PROGRAM Parameters_handler
VAR
	Param_handler:					Data_transforming;
	Handler_floats:					Data_transform_float32;
	Handler_int64:					Data_transform_int64;
END_VAR


// MB_address 40003. PoC nominal Power kVA
Handler_floats(
	Number_variable:= Plant_S_nom, 
	Internal_logic_var:= GVL_PLANT_DEF.Plant_capacity_nom, 
	GUI_var:= GVL_HANDLER.GUI_vars[Plant_S_nom], 
	Modbus_var:= ADR(GVL_HANDLER.Modbus_srv_vars[Plant_S_nom]), 
	RO_RW:= R_O, 
	Min_val:= 0, 
	Max_val:= 3.402823E+38, 
	Def_val:= 8000, 
	Vars_initialization:= GVL_HANDLER.Init_vars, 
	Input_source:= GVL_HANDLER.Input_src,  
	Logic_var_out=> , 
	GUI_var_out=> GVL_HANDLER.GUI_vars[Plant_S_nom]);

// MB_address 40003. PoC nominal voltage
Handler_floats(
	Number_variable:= Plant_V_nom, 
	Internal_logic_var:= GVL_PLANT_DEF.PoC_Voltage_nom, 
	GUI_var:= GVL_HANDLER.GUI_vars[Plant_V_nom], 
	Modbus_var:= ADR(GVL_HANDLER.Modbus_srv_vars[Plant_V_nom]), 
	RO_RW:= R_O, 
	Min_val:= 0, 
	Max_val:= 3.402823E+38, 
	Def_val:= 20000, 
	Vars_initialization:= GVL_HANDLER.Init_vars, 
	Input_source:= GVL_HANDLER.Input_src,  
	Logic_var_out=> , 
	GUI_var_out=> GVL_HANDLER.GUI_vars[Plant_V_nom]);

// MB_address 40005. PoC nominal frequency
Param_handler(
	Number_variable:= Plant_f_nom, 
	GUI_var:= GVL_HANDLER.GUI_vars[Plant_f_nom], 
	Modbus_variable:= GVL_HANDLER.Modbus_srv_vars[Plant_f_nom], 
	Internal_logic_var:= GVL_PLANT_DEF.PoC_freq_nom, 
	RO_RW:= R_W, 
	Scale:= 1, 
	Min_val:= 50, 
	Max_val:= 60, 
	Def_val:= 50, 
	Vars_initialization:= GVL_HANDLER.Init_vars, 
	Input_source:= GVL_HANDLER.Input_src, 
	Logic_var_out=> GVL_PLANT_DEF.PoC_freq_nom, 
	GUI_var_out=> GVL_HANDLER.GUI_vars[Plant_f_nom], 
	Modbus_variable_out=> GVL_HANDLER.Modbus_srv_vars[Plant_f_nom]);
	
// MB_address 40021. N of total converters installed
Param_handler(
	Number_variable:= N_converters, 
	GUI_var:= GVL_HANDLER.GUI_vars[N_converters], 
	Modbus_variable:= GVL_HANDLER.Modbus_srv_vars[N_converters], 
	Internal_logic_var:= WORD_TO_REAL(GVL_CONV_COMMS.NUMBER_CONVERTERS), 
	RO_RW:= R_W, 
	Scale:= 1, 
	Min_val:= 1, 
	Max_val:= 25, 
	Def_val:= 1, 
	Vars_initialization:= GVL_HANDLER.Init_vars, 
	Input_source:= GVL_HANDLER.Input_src, 
	Logic_var_out_wd=> GVL_CONV_COMMS.NUMBER_CONVERTERS,
	GUI_var_out=> GVL_HANDLER.GUI_vars[N_converters], 
	Modbus_variable_out=> GVL_HANDLER.Modbus_srv_vars[N_converters]);
	
// MB_address 40022. nN coefficient. Operative converters over total
Param_handler(
	Number_variable:= nN_converters, 
	GUI_var:= GVL_HANDLER.GUI_vars[nN_converters], 
	Modbus_variable:= GVL_HANDLER.Modbus_srv_vars[nN_converters], 
	Internal_logic_var:= GVL_PLANT_DEF.PoC_freq_nom, 
	RO_RW:= R_O, 
	Scale:= 0.0001, 
	Min_val:= 0, 
	Max_val:= 1, 
	Def_val:= 1, 
	Vars_initialization:= GVL_HANDLER.Init_vars, 
	Input_source:= GVL_HANDLER.Input_src, 
	Logic_var_out=> , 
	GUI_var_out=> GVL_HANDLER.GUI_vars[nN_converters], 
	Modbus_variable_out=> GVL_HANDLER.Modbus_srv_vars[nN_converters]);

// MB_address 40301. P loop type selection
Param_handler(
	Number_variable:= P_loop, 
	GUI_var:= GVL_HANDLER.GUI_vars[P_loop], 
	Modbus_variable:= GVL_HANDLER.Modbus_srv_vars[P_loop], 
	Internal_logic_var:= BOOL_TO_REAL(GVL_P_CONTROL.P_loop_type), 
	RO_RW:= R_W, 
	Scale:= 1, 
	Min_val:= 0, 
	Max_val:= 1, 
	Def_val:= 0, 
	Vars_initialization:= GVL_HANDLER.Init_vars, 
	Input_source:= GVL_HANDLER.Input_src, 
	Logic_var_out_bl=> GVL_P_CONTROL.P_loop_type, 
	GUI_var_out=> GVL_HANDLER.GUI_vars[P_loop], 
	Modbus_variable_out=> GVL_HANDLER.Modbus_srv_vars[P_loop]);
	
// MB_address 40302. P reference 
Param_handler(
	Number_variable:= P_reference, 
	GUI_var:= GVL_HANDLER.GUI_vars[P_reference], 
	Modbus_variable:= GVL_HANDLER.Modbus_srv_vars[P_reference], 
	Internal_logic_var:= GVL_P_CONTROL.P_reference, 
	RO_RW:= R_W, 
	Scale:= 0.01, 
	Min_val:= -100, 
	Max_val:= 100, 
	Def_val:= 1.5, 
	Vars_initialization:= GVL_HANDLER.Init_vars, 
	Input_source:= GVL_HANDLER.Input_src, 
	Logic_var_out=> GVL_P_CONTROL.P_reference, 
	GUI_var_out=> GVL_HANDLER.GUI_vars[P_reference], 
	Modbus_variable_out=> GVL_HANDLER.Modbus_srv_vars[P_reference]);

// MB_address 40303. P feedback 
Param_handler(
	Number_variable:= P_feedback, 
	GUI_var:= GVL_HANDLER.GUI_vars[P_feedback], 
	Modbus_variable:= GVL_HANDLER.Modbus_srv_vars[P_feedback], 
	Internal_logic_var:= GVL_P_CONTROL.P_feedback, 
	RO_RW:= R_O, 
	Scale:= 0.01, 
	Min_val:= -100, 
	Max_val:= 100, 
	Def_val:= 100, 
	Vars_initialization:= GVL_HANDLER.Init_vars, 
	Input_source:= GVL_HANDLER.Input_src, 
	Logic_var_out=> , 
	GUI_var_out=> GVL_HANDLER.GUI_vars[P_feedback], 
	Modbus_variable_out=> GVL_HANDLER.Modbus_srv_vars[P_feedback]);

// MB_address 40304. P output 
Param_handler(
	Number_variable:= P_output, 
	GUI_var:= GVL_HANDLER.GUI_vars[P_output], 
	Modbus_variable:= GVL_HANDLER.Modbus_srv_vars[P_output], 
	Internal_logic_var:= GVL_P_CONTROL.P_output, 
	RO_RW:= R_O, 
	Scale:= 0.01, 
	Min_val:= -100, 
	Max_val:= 100, 
	Def_val:= 100, 
	Vars_initialization:= GVL_HANDLER.Init_vars, 
	Input_source:= GVL_HANDLER.Input_src, 
	Logic_var_out=> , 
	GUI_var_out=> GVL_HANDLER.GUI_vars[P_output], 
	Modbus_variable_out=> GVL_HANDLER.Modbus_srv_vars[P_output]);

// MB_address 40305. P kp 
Param_handler(
	Number_variable:= P_kp, 
	GUI_var:= GVL_HANDLER.GUI_vars[P_kp], 
	Modbus_variable:= GVL_HANDLER.Modbus_srv_vars[P_kp], 
	Internal_logic_var:= GVL_P_CONTROL.P_kp, 
	RO_RW:= R_W, 
	Scale:= 0.001, 
	Min_val:= 0.001, 
	Max_val:= 10, 
	Def_val:= 0.02, 
	Vars_initialization:= GVL_HANDLER.Init_vars, 
	Input_source:= GVL_HANDLER.Input_src, 
	Logic_var_out=> GVL_P_CONTROL.P_kp, 
	GUI_var_out=> GVL_HANDLER.GUI_vars[P_kp], 
	Modbus_variable_out=> GVL_HANDLER.Modbus_srv_vars[P_kp]);

// MB_address 40306. P kp_min 
Param_handler(
	Number_variable:= P_kp_min, 
	GUI_var:= GVL_HANDLER.GUI_vars[P_kp_min], 
	Modbus_variable:= GVL_HANDLER.Modbus_srv_vars[P_kp_min], 
	Internal_logic_var:= GVL_P_CONTROL.P_kp_min, 
	RO_RW:= R_W, 
	Scale:= 0.001, 
	Min_val:= 0.001, 
	Max_val:= 10, 
	Def_val:= 0.02, 
	Vars_initialization:= GVL_HANDLER.Init_vars, 
	Input_source:= GVL_HANDLER.Input_src, 
	Logic_var_out=> GVL_P_CONTROL.P_kp_min, 
	GUI_var_out=> GVL_HANDLER.GUI_vars[P_kp_min], 
	Modbus_variable_out=> GVL_HANDLER.Modbus_srv_vars[P_kp_min]);

// MB_address 40307. P It 
Param_handler(
	Number_variable:= P_ti, 
	GUI_var:= GVL_HANDLER.GUI_vars[P_ti], 
	Modbus_variable:= GVL_HANDLER.Modbus_srv_vars[P_ti], 
	Internal_logic_var:= GVL_P_CONTROL.P_ti, 
	RO_RW:= R_W, 
	Scale:= 0.001, 
	Min_val:= 0.001, 
	Max_val:= 10, 
	Def_val:= 1, 
	Vars_initialization:= GVL_HANDLER.Init_vars, 
	Input_source:= GVL_HANDLER.Input_src, 
	Logic_var_out=> GVL_P_CONTROL.P_ti, 
	GUI_var_out=> GVL_HANDLER.GUI_vars[P_ti], 
	Modbus_variable_out=> GVL_HANDLER.Modbus_srv_vars[P_ti]);

// MB_address 40308. P high anti-windup limit
Param_handler(
	Number_variable:= P_high, 
	GUI_var:= GVL_HANDLER.GUI_vars[P_high], 
	Modbus_variable:= GVL_HANDLER.Modbus_srv_vars[P_high], 
	Internal_logic_var:= GVL_P_CONTROL.P_high_act, 
	RO_RW:= R_W, 
	Scale:= 0.01, 
	Min_val:= 0, 
	Max_val:= 100, 
	Def_val:= 100, 
	Vars_initialization:= GVL_HANDLER.Init_vars, 
	Input_source:= GVL_HANDLER.Input_src, 
	Logic_var_out=> GVL_P_CONTROL.P_high_act, 
	GUI_var_out=> GVL_HANDLER.GUI_vars[P_high], 
	Modbus_variable_out=> GVL_HANDLER.Modbus_srv_vars[P_high]);

// MB_address 40309. P low anti-windup limit
Param_handler(
	Number_variable:= P_low, 
	GUI_var:= GVL_HANDLER.GUI_vars[P_low], 
	Modbus_variable:= GVL_HANDLER.Modbus_srv_vars[P_low], 
	Internal_logic_var:= GVL_P_CONTROL.P_low_act, 
	RO_RW:= R_W, 
	Scale:= 0.01, 
	Min_val:= -100, 
	Max_val:= 0, 
	Def_val:= 0, 
	Vars_initialization:= GVL_HANDLER.Init_vars, 
	Input_source:= GVL_HANDLER.Input_src, 
	Logic_var_out=> GVL_P_CONTROL.P_low_act, 
	GUI_var_out=> GVL_HANDLER.GUI_vars[P_low], 
	Modbus_variable_out=> GVL_HANDLER.Modbus_srv_vars[P_low]);

// MB_address 40310. P PI inversion command
Param_handler(
	Number_variable:= P_invert, 
	GUI_var:= GVL_HANDLER.GUI_vars[P_invert], 
	Modbus_variable:= GVL_HANDLER.Modbus_srv_vars[P_invert], 
	Internal_logic_var:= BOOL_TO_REAL(GVL_P_CONTROL.P_invert), 
	RO_RW:= R_W, 
	Scale:= 1, 
	Min_val:= 0, 
	Max_val:= 1, 
	Def_val:= 0, 
	Vars_initialization:= GVL_HANDLER.Init_vars, 
	Input_source:= GVL_HANDLER.Input_src, 
	Logic_var_out_bl=> GVL_P_CONTROL.P_invert, 
	GUI_var_out=> GVL_HANDLER.GUI_vars[P_invert], 
	Modbus_variable_out=> GVL_HANDLER.Modbus_srv_vars[P_invert]);
	
// MB_address 40311. P to inverters safety position
Param_handler(
	Number_variable:= P_safety, 
	GUI_var:= GVL_HANDLER.GUI_vars[P_safety], 
	Modbus_variable:= GVL_HANDLER.Modbus_srv_vars[P_safety], 
	Internal_logic_var:= GVL_P_CONTROL.P_safety, 
	RO_RW:= R_W, 
	Scale:= 0.01, 
	Min_val:= 0, 
	Max_val:= 100, 
	Def_val:= 0, 
	Vars_initialization:= GVL_HANDLER.Init_vars, 
	Input_source:= GVL_HANDLER.Input_src, 
	Logic_var_out=> GVL_P_CONTROL.P_safety, 
	GUI_var_out=> GVL_HANDLER.GUI_vars[P_safety], 
	Modbus_variable_out=> GVL_HANDLER.Modbus_srv_vars[P_safety]);

// MB_address 40312. P_min indicator
Param_handler(
	Number_variable:= P_min_charge, 
	GUI_var:= GVL_HANDLER.GUI_vars[P_min_charge], 
	Modbus_variable:= GVL_HANDLER.Modbus_srv_vars[P_min_charge], 
	Internal_logic_var:= GVL_POWERMETER.P_min_indicator, 
	RO_RW:= R_O, 
	Scale:= 1, 
	Min_val:= 0, 
	Max_val:= 2, 
	Def_val:= 0, 
	Vars_initialization:= GVL_HANDLER.Init_vars, 
	Input_source:= GVL_HANDLER.Input_src, 
	Logic_var_out=> , 
	GUI_var_out=> GVL_HANDLER.GUI_vars[P_min_charge], 
	Modbus_variable_out=> GVL_HANDLER.Modbus_srv_vars[P_min_charge]);	
	
// MB_address 40501. Q loop type selection
Param_handler(
	Number_variable:= Q_loop, 
	GUI_var:= GVL_HANDLER.GUI_vars[Q_loop], 
	Modbus_variable:= GVL_HANDLER.Modbus_srv_vars[Q_loop], 
	Internal_logic_var:= BOOL_TO_REAL(GVL_Q_CONTROL.Q_loop_type), 
	RO_RW:= R_W, 
	Scale:= 1, 
	Min_val:= 0, 
	Max_val:= 1, 
	Def_val:= 0, 
	Vars_initialization:= GVL_HANDLER.Init_vars, 
	Input_source:= GVL_HANDLER.Input_src, 
	Logic_var_out_bl=> GVL_Q_CONTROL.Q_loop_type, 
	GUI_var_out=> GVL_HANDLER.GUI_vars[Q_loop], 
	Modbus_variable_out=> GVL_HANDLER.Modbus_srv_vars[Q_loop]);
	
// MB_address 40502. Q reference 
Param_handler(
	Number_variable:= Q_reference, 
	GUI_var:= GVL_HANDLER.GUI_vars[Q_reference], 
	Modbus_variable:= GVL_HANDLER.Modbus_srv_vars[Q_reference], 
	Internal_logic_var:= GVL_Q_CONTROL.Q_reference, 
	RO_RW:= R_W, 
	Scale:= 0.01, 
	Min_val:= -100, 
	Max_val:= 100, 
	Def_val:= 0, 
	Vars_initialization:= GVL_HANDLER.Init_vars, 
	Input_source:= GVL_HANDLER.Input_src, 
	Logic_var_out=> GVL_Q_CONTROL.Q_reference, 
	GUI_var_out=> GVL_HANDLER.GUI_vars[Q_reference], 
	Modbus_variable_out=> GVL_HANDLER.Modbus_srv_vars[Q_reference]);

// MB_address 40503. Q feedback 
Param_handler(
	Number_variable:= Q_feedback, 
	GUI_var:= GVL_HANDLER.GUI_vars[Q_feedback], 
	Modbus_variable:= GVL_HANDLER.Modbus_srv_vars[Q_feedback], 
	Internal_logic_var:= GVL_Q_CONTROL.Q_feedback, 
	RO_RW:= R_O, 
	Scale:= 0.01, 
	Min_val:= -100, 
	Max_val:= 100, 
	Def_val:= 100, 
	Vars_initialization:= GVL_HANDLER.Init_vars, 
	Input_source:= GVL_HANDLER.Input_src, 
	Logic_var_out=> , 
	GUI_var_out=> GVL_HANDLER.GUI_vars[Q_feedback], 
	Modbus_variable_out=> GVL_HANDLER.Modbus_srv_vars[Q_feedback]);

// MB_address 40504. Q output 
Param_handler(
	Number_variable:= Q_output, 
	GUI_var:= GVL_HANDLER.GUI_vars[Q_output], 
	Modbus_variable:= GVL_HANDLER.Modbus_srv_vars[Q_output], 
	Internal_logic_var:= GVL_Q_CONTROL.Q_output, 
	RO_RW:= R_O, 
	Scale:= 0.01, 
	Min_val:= -100, 
	Max_val:= 100, 
	Def_val:= 100, 
	Vars_initialization:= GVL_HANDLER.Init_vars, 
	Input_source:= GVL_HANDLER.Input_src, 
	Logic_var_out=> , 
	GUI_var_out=> GVL_HANDLER.GUI_vars[Q_output], 
	Modbus_variable_out=> GVL_HANDLER.Modbus_srv_vars[Q_output]);

// MB_address 40505. Q kQ 
Param_handler(
	Number_variable:= Q_kp, 
	GUI_var:= GVL_HANDLER.GUI_vars[Q_kp], 
	Modbus_variable:= GVL_HANDLER.Modbus_srv_vars[Q_kp], 
	Internal_logic_var:= GVL_Q_CONTROL.Q_kp, 
	RO_RW:= R_W, 
	Scale:= 0.001, 
	Min_val:= 0.001, 
	Max_val:= 10, 
	Def_val:= 0.02, 
	Vars_initialization:= GVL_HANDLER.Init_vars, 
	Input_source:= GVL_HANDLER.Input_src, 
	Logic_var_out=> GVL_Q_CONTROL.Q_kp, 
	GUI_var_out=> GVL_HANDLER.GUI_vars[Q_kp], 
	Modbus_variable_out=> GVL_HANDLER.Modbus_srv_vars[Q_kp]);

// MB_address 40506. Q kp_min 
Param_handler(
	Number_variable:= Q_kp_min, 
	GUI_var:= GVL_HANDLER.GUI_vars[Q_kp_min], 
	Modbus_variable:= GVL_HANDLER.Modbus_srv_vars[Q_kp_min], 
	Internal_logic_var:= GVL_Q_CONTROL.Q_kp_min, 
	RO_RW:= R_W, 
	Scale:= 0.001, 
	Min_val:= 0.001, 
	Max_val:= 10, 
	Def_val:= 0.005, 
	Vars_initialization:= GVL_HANDLER.Init_vars, 
	Input_source:= GVL_HANDLER.Input_src, 
	Logic_var_out=> GVL_Q_CONTROL.Q_kp_min, 
	GUI_var_out=> GVL_HANDLER.GUI_vars[Q_kp_min], 
	Modbus_variable_out=> GVL_HANDLER.Modbus_srv_vars[Q_kp_min]);

// MB_address 40507. Q It 
Param_handler(
	Number_variable:= Q_ti, 
	GUI_var:= GVL_HANDLER.GUI_vars[Q_ti], 
	Modbus_variable:= GVL_HANDLER.Modbus_srv_vars[Q_ti], 
	Internal_logic_var:= GVL_Q_CONTROL.Q_ti, 
	RO_RW:= R_W, 
	Scale:= 0.001, 
	Min_val:= 0.001, 
	Max_val:= 10, 
	Def_val:= 1, 
	Vars_initialization:= GVL_HANDLER.Init_vars, 
	Input_source:= GVL_HANDLER.Input_src, 
	Logic_var_out=> GVL_Q_CONTROL.Q_ti, 
	GUI_var_out=> GVL_HANDLER.GUI_vars[Q_ti], 
	Modbus_variable_out=> GVL_HANDLER.Modbus_srv_vars[Q_ti]);

// MB_address 40508. Q high anti-winduQ limit
Param_handler(
	Number_variable:= Q_high, 
	GUI_var:= GVL_HANDLER.GUI_vars[Q_high], 
	Modbus_variable:= GVL_HANDLER.Modbus_srv_vars[Q_high], 
	Internal_logic_var:= GVL_Q_CONTROL.Q_high_act, 
	RO_RW:= R_W, 
	Scale:= 0.01, 
	Min_val:= 0, 
	Max_val:= 100, 
	Def_val:= 100, 
	Vars_initialization:= GVL_HANDLER.Init_vars, 
	Input_source:= GVL_HANDLER.Input_src, 
	Logic_var_out=> GVL_Q_CONTROL.Q_high_act, 
	GUI_var_out=> GVL_HANDLER.GUI_vars[Q_high], 
	Modbus_variable_out=> GVL_HANDLER.Modbus_srv_vars[Q_high]);

// MB_address 40509. Q low anti-winduQ limit
Param_handler(
	Number_variable:= Q_low, 
	GUI_var:= GVL_HANDLER.GUI_vars[Q_low], 
	Modbus_variable:= GVL_HANDLER.Modbus_srv_vars[Q_low], 
	Internal_logic_var:= GVL_Q_CONTROL.Q_low_act, 
	RO_RW:= R_W, 
	Scale:= 0.01, 
	Min_val:= -100, 
	Max_val:= 0, 
	Def_val:= 0, 
	Vars_initialization:= GVL_HANDLER.Init_vars, 
	Input_source:= GVL_HANDLER.Input_src, 
	Logic_var_out=> GVL_Q_CONTROL.Q_low_act, 
	GUI_var_out=> GVL_HANDLER.GUI_vars[Q_low], 
	Modbus_variable_out=> GVL_HANDLER.Modbus_srv_vars[Q_low]);

// MB_address 40510. Q PI inversion command
Param_handler(
	Number_variable:= Q_invert, 
	GUI_var:= GVL_HANDLER.GUI_vars[Q_invert], 
	Modbus_variable:= GVL_HANDLER.Modbus_srv_vars[Q_invert], 
	Internal_logic_var:= BOOL_TO_REAL(GVL_Q_CONTROL.Q_invert), 
	RO_RW:= R_W, 
	Scale:= 1, 
	Min_val:= 0, 
	Max_val:= 1, 
	Def_val:= 0, 
	Vars_initialization:= GVL_HANDLER.Init_vars, 
	Input_source:= GVL_HANDLER.Input_src, 
	Logic_var_out_bl=> GVL_Q_CONTROL.Q_invert, 
	GUI_var_out=> GVL_HANDLER.GUI_vars[Q_invert], 
	Modbus_variable_out=> GVL_HANDLER.Modbus_srv_vars[Q_invert]);
	
// MB_address 40511. Q to inverters safety position
Param_handler(
	Number_variable:= Q_safety, 
	GUI_var:= GVL_HANDLER.GUI_vars[Q_safety], 
	Modbus_variable:= GVL_HANDLER.Modbus_srv_vars[Q_safety], 
	Internal_logic_var:= GVL_Q_CONTROL.Q_safety, 
	RO_RW:= R_W, 
	Scale:= 0.01, 
	Min_val:= 0, 
	Max_val:= 100, 
	Def_val:= 0, 
	Vars_initialization:= GVL_HANDLER.Init_vars, 
	Input_source:= GVL_HANDLER.Input_src, 
	Logic_var_out=> GVL_Q_CONTROL.Q_safety, 
	GUI_var_out=> GVL_HANDLER.GUI_vars[Q_safety], 
	Modbus_variable_out=> GVL_HANDLER.Modbus_srv_vars[Q_safety]);

// MB_address 40512. Q ramps enable
Param_handler(
	Number_variable:= Ramp_enable, 
	GUI_var:= GVL_HANDLER.GUI_vars[Ramp_enable], 
	Modbus_variable:= GVL_HANDLER.Modbus_srv_vars[Ramp_enable], 
	Internal_logic_var:= BOOL_TO_REAL(GVL_Q_CONTROL.Ramp_enable), 
	RO_RW:= R_W, 
	Scale:= 1, 
	Min_val:= 0, 
	Max_val:= 1, 
	Def_val:= 0, 
	Vars_initialization:= GVL_HANDLER.Init_vars, 
	Input_source:= GVL_HANDLER.Input_src, 
	Logic_var_out_bl=> GVL_Q_CONTROL.Ramp_enable, 
	GUI_var_out=> GVL_HANDLER.GUI_vars[Ramp_enable], 
	Modbus_variable_out=> GVL_HANDLER.Modbus_srv_vars[Ramp_enable]);
	
// MB_address 40513. Q ramps time elapsed ramping 
Param_handler(
	Number_variable:= Time_span, 
	GUI_var:= GVL_HANDLER.GUI_vars[Time_span], 
	Modbus_variable:= GVL_HANDLER.Modbus_srv_vars[Time_span], 
	Internal_logic_var:= GVL_Q_CONTROL.Time_span, 
	RO_RW:= R_O, 
	Scale:= 1, 
	Min_val:= 1, 
	Max_val:= 1, 
	Def_val:= 3600, 
	Vars_initialization:= GVL_HANDLER.Init_vars, 
	Input_source:= GVL_HANDLER.Input_src, 
	Logic_var_out=> , 
	GUI_var_out=> GVL_HANDLER.GUI_vars[Time_span], 
	Modbus_variable_out=> GVL_HANDLER.Modbus_srv_vars[Time_span]);

// MB_address 40514. Q increasing ramp value
Param_handler(
	Number_variable:= R_up_value, 
	GUI_var:= GVL_HANDLER.GUI_vars[R_up_value], 
	Modbus_variable:= GVL_HANDLER.Modbus_srv_vars[R_up_value], 
	Internal_logic_var:= GVL_Q_CONTROL.Ramp_up_value, 
	RO_RW:= R_W, 
	Scale:= 0.01, 
	Min_val:= 0, 
	Max_val:= 655.35, 
	Def_val:= 0, 
	Vars_initialization:= GVL_HANDLER.Init_vars, 
	Input_source:= GVL_HANDLER.Input_src, 
	Logic_var_out=> GVL_Q_CONTROL.Ramp_up_value, 
	GUI_var_out=> GVL_HANDLER.GUI_vars[R_up_value], 
	Modbus_variable_out=> GVL_HANDLER.Modbus_srv_vars[R_up_value]);

// MB_address 40515. Q decreasing ramp value
Param_handler(
	Number_variable:= R_down_value, 
	GUI_var:= GVL_HANDLER.GUI_vars[R_down_value], 
	Modbus_variable:= GVL_HANDLER.Modbus_srv_vars[R_down_value], 
	Internal_logic_var:= GVL_Q_CONTROL.Ramp_down_value, 
	RO_RW:= R_W, 
	Scale:= 0.01, 
	Min_val:= 0, 
	Max_val:= 655.35, 
	Def_val:= 0, 
	Vars_initialization:= GVL_HANDLER.Init_vars, 
	Input_source:= GVL_HANDLER.Input_src, 
	Logic_var_out=> GVL_Q_CONTROL.Ramp_down_value, 
	GUI_var_out=> GVL_HANDLER.GUI_vars[R_down_value], 
	Modbus_variable_out=> GVL_HANDLER.Modbus_srv_vars[R_down_value]);

// MB_address 40516. Q ramps units enumeration
Param_handler(
	Number_variable:= R_units, 
	GUI_var:= GVL_HANDLER.GUI_vars[R_units], 
	Modbus_variable:= GVL_HANDLER.Modbus_srv_vars[R_units], 
	Internal_logic_var:= WORD_TO_REAL(GVL_Q_CONTROL.Ramp_units), 
	RO_RW:= R_W, 
	Scale:= 1, 
	Min_val:= 1, 
	Max_val:= 25, 
	Def_val:= 1, 
	Vars_initialization:= GVL_HANDLER.Init_vars, 
	Input_source:= GVL_HANDLER.Input_src, 
	Logic_var_out_wd=> GVL_Q_CONTROL.Ramp_units,
	GUI_var_out=> GVL_HANDLER.GUI_vars[R_units], 
	Modbus_variable_out=> GVL_HANDLER.Modbus_srv_vars[R_units]);
	
// MB_address 41201. Active positive energy in kWh
Handler_int64(
	Number_variable:= Active_er_pos_kWh, 
	Internal_logic_var:= GVL_POWERMETER.Active_er_pos_kWh, 
	GUI_var:= REAL_TO_LINT(GVL_HANDLER.GUI_vars[Active_er_pos_kWh]), 
	MB_variable:= ADR(GVL_HANDLER.Modbus_srv_vars[Active_er_pos_kWh]), 
	RO_RW:= R_O, 
	Min_val:= -9223372036854775808, 
	Max_val:= 9223372036854775807, 
	Def_val:= 0, 
	Vars_initialization:= GVL_HANDLER.Init_vars, 
	Input_source:= GVL_HANDLER.Input_src,  
	Logic_var_int64_out=> , 
	GUI_var_out=> GVL_HANDLER.GUI_vars[Active_er_pos_kWh]);
	
// MB_address 41205. Active negative energy in kWh
Handler_int64(
	Number_variable:= Active_er_neg_kWh, 
	Internal_logic_var:= GVL_POWERMETER.Active_er_neg_kWh, 
	GUI_var:= REAL_TO_LINT(GVL_HANDLER.GUI_vars[Active_er_neg_kWh]), 
	MB_variable:= ADR(GVL_HANDLER.Modbus_srv_vars[Active_er_neg_kWh]), 
	RO_RW:= R_O, 
	Min_val:= -9223372036854775808, 
	Max_val:= 9223372036854775807, 
	Def_val:= 0, 
	Vars_initialization:= GVL_HANDLER.Init_vars, 
	Input_source:= GVL_HANDLER.Input_src,  
	Logic_var_int64_out=> , 
	GUI_var_out=> GVL_HANDLER.GUI_vars[Active_er_neg_kWh]);
	
// MB_address 41209. Active energy total in kWh
Handler_int64(
	Number_variable:= Active_er_tot_kWh, 
	Internal_logic_var:= GVL_POWERMETER.Active_er_tot_kWh, 
	GUI_var:= REAL_TO_LINT(GVL_HANDLER.GUI_vars[Active_er_tot_kWh]), 
	MB_variable:= ADR(GVL_HANDLER.Modbus_srv_vars[Active_er_tot_kWh]), 
	RO_RW:= R_O, 
	Min_val:= -9223372036854775808, 
	Max_val:= 9223372036854775807, 
	Def_val:= 0, 
	Vars_initialization:= GVL_HANDLER.Init_vars, 
	Input_source:= GVL_HANDLER.Input_src,  
	Logic_var_int64_out=> , 
	GUI_var_out=> GVL_HANDLER.GUI_vars[Active_er_tot_kWh]);

// MB_address 41213. Rective positive energy in kVArh
Handler_int64(
	Number_variable:= React_er_pos_kVArh, 
	Internal_logic_var:= GVL_POWERMETER.React_er_pos_kVArh, 
	GUI_var:= REAL_TO_LINT(GVL_HANDLER.GUI_vars[React_er_pos_kVArh]), 
	MB_variable:= ADR(GVL_HANDLER.Modbus_srv_vars[React_er_pos_kVArh]), 
	RO_RW:= R_O, 
	Min_val:= -9223372036854775808, 
	Max_val:= 9223372036854775807, 
	Def_val:= 0, 
	Vars_initialization:= GVL_HANDLER.Init_vars, 
	Input_source:= GVL_HANDLER.Input_src,  
	Logic_var_int64_out=> , 
	GUI_var_out=> GVL_HANDLER.GUI_vars[React_er_pos_kVArh]);

// MB_address 41213. Rective negative energy in kVArh
Handler_int64(
	Number_variable:= React_er_neg_kVArh, 
	Internal_logic_var:= GVL_POWERMETER.React_er_neg_kVArh, 
	GUI_var:= REAL_TO_LINT(GVL_HANDLER.GUI_vars[React_er_neg_kVArh]), 
	MB_variable:= ADR(GVL_HANDLER.Modbus_srv_vars[React_er_neg_kVArh]), 
	RO_RW:= R_O, 
	Min_val:= -9223372036854775808, 
	Max_val:= 9223372036854775807, 
	Def_val:= 0, 
	Vars_initialization:= GVL_HANDLER.Init_vars, 
	Input_source:= GVL_HANDLER.Input_src,  
	Logic_var_int64_out=> , 
	GUI_var_out=> GVL_HANDLER.GUI_vars[React_er_neg_kVArh]);

// MB_address 41213. Rective energy total in kVArh
Handler_int64(
	Number_variable:= React_er_tot_kVArh, 
	Internal_logic_var:= GVL_POWERMETER.React_er_tot_kVArh, 
	GUI_var:= REAL_TO_LINT(GVL_HANDLER.GUI_vars[React_er_tot_kVArh]), 
	MB_variable:= ADR(GVL_HANDLER.Modbus_srv_vars[React_er_tot_kVArh]), 
	RO_RW:= R_O, 
	Min_val:= -9223372036854775808, 
	Max_val:= 9223372036854775807, 
	Def_val:= 0, 
	Vars_initialization:= GVL_HANDLER.Init_vars, 
	Input_source:= GVL_HANDLER.Input_src,  
	Logic_var_int64_out=> , 
	GUI_var_out=> GVL_HANDLER.GUI_vars[React_er_tot_kVArh]);
	
// MB_address 41225. Energies counter reset
Param_handler(
	Number_variable:= Energies_reset, 
	GUI_var:= GVL_HANDLER.GUI_vars[Energies_reset], 
	Modbus_variable:= GVL_HANDLER.Modbus_srv_vars[Energies_reset], 
	Internal_logic_var:= BOOL_TO_REAL(GVL_POWERMETER.Energies_reset), 
	RO_RW:= R_W, 
	Scale:= 1, 
	Min_val:= 0, 
	Max_val:= 1, 
	Def_val:= 0, 
	Vars_initialization:= GVL_HANDLER.Init_vars, 
	Input_source:= GVL_HANDLER.Input_src, 
	Logic_var_out_bl=> GVL_POWERMETER.Energies_reset, 
	GUI_var_out=> GVL_HANDLER.GUI_vars[Energies_reset], 
	Modbus_variable_out=> GVL_HANDLER.Modbus_srv_vars[Energies_reset]);
	
// MB_address 41131. Meter board status
Param_handler(
	Number_variable:= Meter_status, 
	GUI_var:= GVL_HANDLER.GUI_vars[Meter_status], 
	Modbus_variable:= GVL_HANDLER.Modbus_srv_vars[Meter_status], 
	Internal_logic_var:= BOOL_TO_REAL(GVL_POWERMETER.Meter_comms_status), 
	RO_RW:= R_O, 
	Scale:= 1, 
	Min_val:= 1, 
	Max_val:= 25, 
	Def_val:= 1, 
	Vars_initialization:= GVL_HANDLER.Init_vars, 
	Input_source:= GVL_HANDLER.Input_src, 
	Logic_var_out_bl=> ,
	GUI_var_out=> GVL_HANDLER.GUI_vars[Meter_status], 
	Modbus_variable_out=> GVL_HANDLER.Modbus_srv_vars[Meter_status]);

// MB_address 41132. Meter lost comms algorithm enable
Param_handler(
	Number_variable:= Lost_comms_enable, 
	GUI_var:= GVL_HANDLER.GUI_vars[Lost_comms_enable], 
	Modbus_variable:= GVL_HANDLER.Modbus_srv_vars[Lost_comms_enable], 
	Internal_logic_var:= BOOL_TO_REAL(GVL_POWERMETER.Alg_lost_comms_enable), 
	RO_RW:= R_W, 
	Scale:= 1, 
	Min_val:= 0, 
	Max_val:= 1, 
	Def_val:= 0, 
	Vars_initialization:= GVL_HANDLER.Init_vars, 
	Input_source:= GVL_HANDLER.Input_src, 
	Logic_var_out_bl=> GVL_POWERMETER.Alg_lost_comms_enable, 
	GUI_var_out=> GVL_HANDLER.GUI_vars[Lost_comms_enable], 
	Modbus_variable_out=> GVL_HANDLER.Modbus_srv_vars[Lost_comms_enable]);

// MB_address 41201. V trfr measures RS
Handler_floats(
	Number_variable:= V_ratio_RS, 
	Internal_logic_var:= GVL_PM_CONFIG.Voltage_trafo_rat_L1, 
	GUI_var:= GVL_HANDLER.GUI_vars[V_ratio_RS], 
	Modbus_var:= ADR(GVL_HANDLER.Modbus_srv_vars[V_ratio_RS]), 
	RO_RW:= R_W, 
	Min_val:= -3.402823E+38, 
	Max_val:= 3.402823E+38, 
	Def_val:= 1, 
	Vars_initialization:= GVL_HANDLER.Init_vars, 
	Input_source:= GVL_HANDLER.Input_src,  
	Logic_var_out=> , 
	GUI_var_out=> GVL_HANDLER.GUI_vars[V_ratio_RS]);
	
// MB_address 41203. V trfr measures ST
Handler_floats(
	Number_variable:= V_ratio_ST, 
	Internal_logic_var:= GVL_PM_CONFIG.Voltage_trafo_rat_L2, 
	GUI_var:= GVL_HANDLER.GUI_vars[V_ratio_ST], 
	Modbus_var:= ADR(GVL_HANDLER.Modbus_srv_vars[V_ratio_ST]), 
	RO_RW:= R_W, 
	Min_val:= -3.402823E+38, 
	Max_val:= 3.402823E+38, 
	Def_val:= 1, 
	Vars_initialization:= GVL_HANDLER.Init_vars, 
	Input_source:= GVL_HANDLER.Input_src,  
	Logic_var_out=> , 
	GUI_var_out=> GVL_HANDLER.GUI_vars[V_ratio_ST]);
	
// MB_address 41205. V trfr measures RS
Handler_floats(
	Number_variable:= V_ratio_TR, 
	Internal_logic_var:= GVL_PM_CONFIG.Voltage_trafo_rat_L3, 
	GUI_var:= GVL_HANDLER.GUI_vars[V_ratio_TR], 
	Modbus_var:= ADR(GVL_HANDLER.Modbus_srv_vars[V_ratio_TR]), 
	RO_RW:= R_W, 
	Min_val:= -3.402823E+38, 
	Max_val:= 3.402823E+38, 
	Def_val:= 1, 
	Vars_initialization:= GVL_HANDLER.Init_vars, 
	Input_source:= GVL_HANDLER.Input_src,  
	Logic_var_out=> , 
	GUI_var_out=> GVL_HANDLER.GUI_vars[V_ratio_TR]);

// MB_address 41207. I trfr measures ratio R
Handler_floats(
	Number_variable:= I_ratio_R, 
	Internal_logic_var:= GVL_PM_CONFIG.Current_trafo_rat_L1, 
	GUI_var:= GVL_HANDLER.GUI_vars[I_ratio_R], 
	Modbus_var:= ADR(GVL_HANDLER.Modbus_srv_vars[I_ratio_R]), 
	RO_RW:= R_W, 
	Min_val:= -3.402823E+38, 
	Max_val:= 3.402823E+38, 
	Def_val:= 1, 
	Vars_initialization:= GVL_HANDLER.Init_vars, 
	Input_source:= GVL_HANDLER.Input_src,  
	Logic_var_out=> , 
	GUI_var_out=> GVL_HANDLER.GUI_vars[I_ratio_R]);

// MB_address 41209. I trfr measures ratio S
Handler_floats(
	Number_variable:= I_ratio_S, 
	Internal_logic_var:= GVL_PM_CONFIG.Current_trafo_rat_L2, 
	GUI_var:= GVL_HANDLER.GUI_vars[I_ratio_S], 
	Modbus_var:= ADR(GVL_HANDLER.Modbus_srv_vars[I_ratio_S]), 
	RO_RW:= R_W, 
	Min_val:= -3.402823E+38, 
	Max_val:= 3.402823E+38, 
	Def_val:= 1, 
	Vars_initialization:= GVL_HANDLER.Init_vars, 
	Input_source:= GVL_HANDLER.Input_src,  
	Logic_var_out=> , 
	GUI_var_out=> GVL_HANDLER.GUI_vars[I_ratio_S]);

// MB_address 41211. I trfr measures ratio T
Handler_floats(
	Number_variable:= I_ratio_T, 
	Internal_logic_var:= GVL_PM_CONFIG.Current_trafo_rat_L3, 
	GUI_var:= GVL_HANDLER.GUI_vars[I_ratio_T], 
	Modbus_var:= ADR(GVL_HANDLER.Modbus_srv_vars[I_ratio_T]), 
	RO_RW:= R_W, 
	Min_val:= -3.402823E+38, 
	Max_val:= 3.402823E+38, 
	Def_val:= 1, 
	Vars_initialization:= GVL_HANDLER.Init_vars, 
	Input_source:= GVL_HANDLER.Input_src,  
	Logic_var_out=> , 
	GUI_var_out=> GVL_HANDLER.GUI_vars[I_ratio_T]);

END_PROGRAM

// ---- POUs/HANDLER_PARAM/Data_transforming.TcPOU
FUNCTION_BLOCK Data_transforming
VAR_INPUT
	Number_variable: 			INT;
	GUI_var: 					REAL;
	Modbus_variable: 			WORD;
	Internal_logic_var:			REAL;
	RO_RW: 						INT;
	Scale: 						REAL;
	Min_val: 					REAL;
	Max_val: 					REAL;
	Def_val: 					REAL;
	Vars_initialization:		BOOL;
	Input_source:				BOOL; //TRUE -> Modbus, FALSE -> Web GUI
END_VAR

VAR_OUTPUT
	Logic_var_out: 				REAL;
	Logic_var_out_wd: 			WORD;
	Logic_var_out_bl: 			BOOL;
	
	GUI_var_out: 				REAL;
	Modbus_variable_out: 		WORD;
END_VAR	

VAR
	Modbus_var_internal : 		REAL;
	
END_VAR

(*
***************************************************************************************************

Function to control the process variable from WEBSERVER or MODBUS. Also applies scales for the MB

*****************************************************************************************************
*)

// First of all, it is necessary to know if the variable is read or write
IF RO_RW = R_W THEN
	
		// Check if the control is by webserver or by Modbus (in this case webserver)
		IF NOT Input_source THEN
			
			// Compare if the web variable is different than the process variable
			IF GUI_var <> Internal_logic_var THEN
				// Checking if the new value is within the range.
				IF 	GUI_var >= Min_val AND GUI_var <= Max_val THEN
					Internal_logic_var := GUI_var;
				ELSE
					GUI_var := Internal_logic_var;
				END_IF
			END_IF
		ELSE
			// When the control is by Modbus apply scaling for decimal figures
			Modbus_var_internal := (WORD_TO_INT(Modbus_variable)) * Scale;
			// Compare if the Modbus variable is different than the process variable
			IF Modbus_var_internal <> Internal_logic_var THEN
				// Checking if the new value is within the range
				IF 	Modbus_var_internal > Min_val AND Modbus_var_internal < Max_val THEN
					Internal_logic_var := Modbus_var_internal;
				ELSE
					Modbus_var_internal := Internal_logic_var;
				END_IF
			
			END_IF
			
		END_IF
	ELSE
	
		Modbus_var_internal := Internal_logic_var;
		GUI_var := Internal_logic_var;
	
END_IF

//////////////////////////////////////////////////////////////////////////////////////////////////////////////////////////////////////////////////

(*
IF R_W_mode = R_W_STATUS THEN
	
	Proces_Variable_Word:= REAL_TO_WORD(Internal_logic_var);

	Byte_Web_Variable:= REAL_TO_BYTE(GUI_var);
	Byte_Modbus_Variable:= REAL_TO_BYTE(Modbus_variable);
	
	BYTE_EXTRACTION_1(	Divisible_Word:= Proces_Variable_Word,
						Upper:= FALSE,
						Selected_Byte=> Control_Byte,
					 );
	
	BYTE_EXTRACTION_2(	Divisible_Word:= Proces_Variable_Word,
						Upper:= TRUE,
						Selected_Byte=> Status_Byte,
					 );	

					
	
	IF Data_Handling.Init_Data_Handling = FALSE THEN
	
		// Check if the control is by webserver or by Modbus (in this case webserver)
		IF COMMS_VAR.Control_COMMS = 0 THEN
			
			// Compare if the web variable is different than the process variable
			IF Byte_Web_variable <> Control_Byte THEN
				
				// Registering of the parameter that is going to be modified
				//Data_Handling_VAR.Parameter_recording[USER] := ;
				Data_Handling_VAR.Parameter_recording[PARAMETER_NUMBER] := Number_variable;
				Data_Handling_VAR.Parameter_recording[OLD_VALUE] := BYTE_TO_REAL (Control_Byte);
				Data_Handling_VAR.Parameter_recording_String := Description;
			
				// Checking if the new value is withing the range. Is adding +/- scale because the decimal 
				IF 	Byte_Web_Variable >= Min_val AND Byte_Web_Variable <= Max_val THEN
					Control_Byte := Byte_Web_Variable;
				ELSE
					Byte_Web_Variable := Control_Byte;
				END_IF
				
				// Record the new value modified
				Data_Handling_VAR.Parameter_recording[NEW_VALUE] := BYTE_TO_REAL(Byte_Web_Variable);
			
			END_IF
			
		ELSE
		
			// When the control is by Modbus, first of all, it is necessary scale the Modbus Variable
			Modbus_Byte := Byte_Modbus_Variable;
			
			// Compare if the Modbus variable is different than the process variable
			IF Modbus_Byte <> Control_Byte THEN
				
				// Registering of the parameter that is going to be modified
				//Data_Handling_VAR.Parameter_recording[USER] := ;
				Data_Handling_VAR.Parameter_recording[PARAMETER_NUMBER] := Number_variable;
				Data_Handling_VAR.Parameter_recording[OLD_VALUE] := BYTE_TO_REAL(Control_Byte);
				Data_Handling_VAR.Parameter_recording_String := Description;
			
				// Checking if the new value is withing the range. Is adding +/- scale because the decimal 
				IF 	Modbus_Byte >= Min_val AND Modbus_Byte <= Max_val THEN
					Control_Byte := Modbus_Byte;
				ELSE
					Modbus_Byte := Control_Byte;
				END_IF
				
				// Record the new value modified
				Data_Handling_VAR.Parameter_recording[NEW_VALUE] := BYTE_TO_REAL(Control_Byte);
			
			END_IF
			
		END_IF
	ELSE
	
		Modbus_var_internal := Internal_logic_var;
		GUI_var := Internal_logic_var;
		
		
		
	END_IF
	
	BYTE_UNION_1(	Upper_Byte:= Status_Byte,
					Lower_Byte:= Control_Byte,
					United_Word=> Proces_Variable_Word);

	Internal_logic_var:= WORD_TO_REAL(Proces_Variable_Word);
	
	
END_IF
*)

//////////////////////////////////////////////////////////////////////////////////////////////////////////////////////////////////////////////////

	// Finally, either Read or Read/Write, and not Read/Write Word, logic variable is written in the Modbus and GUI
	Logic_var_out:= Internal_logic_var;
	Logic_var_out_wd:= REAL_TO_WORD(Internal_logic_var);
	Logic_var_out_bl:= REAL_TO_BOOL(Internal_logic_var);
	
	GUI_var_out := Internal_logic_var;
	Modbus_variable_out := REAL_TO_WORD(Internal_logic_var / scale);
	
// When the user do a initialization, all variables takes the default value
IF Vars_initialization THEN
	Logic_var_out := Def_val;
	Logic_var_out_wd:= REAL_TO_WORD(Def_val);
	Logic_var_out_bl:= REAL_TO_BOOL(Def_val);
	
	GUI_var_out := Def_val;
	Modbus_variable_out := REAL_TO_WORD(Def_val / Scale);
END_IF

END_FUNCTION_BLOCK

// ---- POUs/HANDLER_PARAM/Data_transform_float32.TcPOU
FUNCTION_BLOCK Data_transform_float32
VAR_INPUT
	Number_variable: 				INT;
	Internal_logic_var: 			REAL;
	GUI_var: 						REAL;
	Modbus_var: 					POINTER TO BYTE;
	RO_RW: 							INT;
	Min_val: 						REAL;
	Max_val: 						REAL;
	Def_val: 						REAL;
	Vars_initialization:			BOOL;
	Input_source:					BOOL; //TRUE -> Modbus, FALSE -> Web GUI
END_VAR

VAR_OUTPUT
	Logic_var_out: 					REAL;
	GUI_var_out: 					REAL;
END_VAR

VAR
	Pt_REAL: 						POINTER TO REAL;
	Aux_REAL:						REAL; 
END_VAR

// First of all, it is necessary to know if the variable is read or write
IF RO_RW = R_W THEN
	// Check if the control is by Web GUI or by Modbus (in this case webserver)
	IF NOT Input_source THEN
		
	// Compare if the web variable is different than the process variable
		IF GUI_var <> Internal_logic_var THEN
			// Checking if the new value is within the range.
			IF 	GUI_var > Min_val AND GUI_var < Max_val THEN
				Internal_logic_var := GUI_var;
			ELSE
				GUI_var := Internal_logic_var;
			END_IF
		END_IF
	ELSE
		// Obtaining the real
		Pt_REAL:= Modbus_var;
		Aux_REAL:= Pt_REAL^;
		
		// Compare if the Modbus variable is different than the logic variable
		IF Aux_REAL <> Internal_logic_var THEN
			// Checking if the new value is within the range.
			IF 	Aux_REAL > Min_val AND Aux_REAL < Max_val THEN
				Internal_logic_var := Aux_REAL;
			ELSE
				Aux_REAL := Internal_logic_var;
			END_IF
		END_IF
	END_IF
ELSE
	Aux_REAL := Internal_logic_var;
	GUI_var := Internal_logic_var;
END_IF

Logic_var_out:= Internal_logic_var;
GUI_var_out := Internal_logic_var;
MEMMOVE(destAddr:= Modbus_var, srcAddr:= ADR(Internal_logic_var), n:= SIZEOF(Internal_logic_var));
	
// When the user do a initialization, all variables take default value
IF Vars_initialization THEN
	Logic_var_out := Def_val;
	GUI_var_out := Def_val;
	MEMMOVE(destAddr:= Modbus_var, srcAddr:= ADR(Def_val), n:= SIZEOF(Def_val));
END_IF

END_FUNCTION_BLOCK

// ---- POUs/HANDLER_PARAM/Data_transform_int64.TcPOU
FUNCTION_BLOCK Data_transform_int64
VAR_INPUT
	Number_variable: 				INT;
	Internal_logic_var: 			LINT;
	GUI_var: 						LINT;
	MB_variable: 					POINTER TO BYTE;
	RO_RW: 							INT;
	Min_val: 						LINT;
	Max_val: 						LINT;
	Def_val: 						LINT;
	Vars_initialization:			BOOL;
	Input_source:					BOOL; //TRUE -> Modbus, FALSE -> Web GUI

END_VAR

VAR_OUTPUT
	Logic_var_int64_out: 			LINT;
	GUI_var_out: 					REAL;
END_VAR

VAR
	Pt_LINT: 						POINTER TO LINT;
	Aux_LINT:						LINT; 
	
	R_W_Mode_String: 				STRING;
	
	Debug_Scale: 					INT:= 1;
END_VAR

IF RO_RW = R_W THEN
	IF NOT Input_source THEN
		// Compare if the web variable is different than the process variable
		IF GUI_var <> Internal_logic_var THEN
			// Checking if the new value is withing the range. Is adding +/- scale because the decimal 
			IF 	GUI_var > Min_val AND GUI_var < Max_val THEN
				Internal_logic_var := GUI_var;
			ELSE
				GUI_var := Internal_logic_var;
			END_IF
		END_IF
	ELSE
		Pt_LINT:= MB_variable;
		Aux_LINT:= Pt_LINT^;		
		// Compare if the modbus variable is different
		IF Aux_LINT <> Internal_logic_var THEN		
			// Checking if the new value is withing the range.  
			IF 	Aux_LINT > Min_val AND Aux_LINT < Max_val THEN
				Internal_logic_var := Aux_LINT;
			ELSE
				Aux_LINT := Internal_logic_var;
			END_IF
		END_IF
	END_IF
ELSE
	Aux_LINT := Internal_logic_var;
	GUI_var := Internal_logic_var;
END_IF

// Finally, either Read or Read/Write, and not Read/Write Word, the logic variable is written in the Modbus and Web GUI
Logic_var_int64_out:= Internal_logic_var;
GUI_var_out := LINT_TO_REAL(Internal_logic_var);
MEMCPY(destAddr:= MB_variable, srcAddr:= ADR(Internal_logic_var), n:= SIZEOF(Internal_logic_var));
	
// If initialization is done, all variables take def value
IF Vars_initialization THEN
	Logic_var_int64_out := Def_val;
	GUI_var_out := LINT_TO_REAL(Def_val);
	MEMCPY(destAddr:= MB_variable, srcAddr:= ADR(Def_val), n:= SIZEOF(Def_val));	
END_IF

END_FUNCTION_BLOCK

// ---- POUs/BYTE_UNION.TcPOU
FUNCTION_BLOCK BYTE_UNION

VAR_INPUT
	Upper_Byte:			BYTE;
	Lower_Byte:			BYTE;
END_VAR

VAR_OUTPUT
	United_Word:		WORD;
END_VAR

VAR
	Aux_Word:			WORD;
END_VAR

Aux_Word:= BYTE_TO_WORD (Upper_Byte);
United_Word:= SHL (Aux_Word, 8) + Lower_Byte;

END_FUNCTION_BLOCK

// ---- POUs/VISU_HANDLER/GUI_logic.TcPOU
PROGRAM GUI_logic
VAR
END_VAR

(*
//Main screen GUI buttons
IF GVL_GUI.main_button_logic THEN
	GVL_GUI.conv_button_logic:= 0;
	GVL_GUI.pcontrol_button_logic:= 0;
	GVL_GUI.qcontrol_button_logic:= 0;
	GVL_GUI.meter_cfg_button_logic:= 0;
ELSIF GVL_GUI.pcontrol_button_logic THEN
	GVL_GUI.main_button_logic:= 0;
	GVL_GUI.conv_button_logic:= 0;
	GVL_GUI.qcontrol_button_logic:= 0;
	GVL_GUI.meter_cfg_button_logic:= 0;
ELSE
	GVL_GUI.main_button_logic:= 0;
	GVL_GUI.conv_button_logic:= 0;
	GVL_GUI.pcontrol_button_logic:= 0;
	GVL_GUI.qcontrol_button_logic:= 0;
	GVL_GUI.meter_cfg_button_logic:= 0;
END_IF
*)

END_PROGRAM

// ---- GlobalTextList.TcGTLO
TEXTLIST GlobalTextList
  408 = ' invert PI'
  481 = '%%.1f kW%'
  612 = '%%.2f %'
  37 = '%.1f'
  225 = '%.1f kVAr'
  297 = '%.1f kW'
  75 = '%.1f kW%'
  250 = '%.1fkVAr'
  457 = '%.2d kVA'
  143 = '%.2f'
  848 = '%.2f %%'
  989 = '%.2f kVA'
  459 = '%.2f kW'
  238 = '%.3f'
  468 = '%.3f kVA'
  824 = '%.3f kVAr'
  667 = '%.3f kW'
  633 = '%.3f V'
  1112 = '%d kVA'
  942 = '%d kVAr'
  637 = '%d kVArh'
  422 = '%d kW'
  393 = '%d kWh'
  101 = '%f.3'
  239 = '%s'
  148 = '+'
  901 = '-'
  955 = '0°'
  4316 = '120°'
  1928 = '150°'
  2469 = '180°'
  674 = '192.168.254.32'
  1336 = '210°'
  1219 = '240°'
  4647 = '270°'
  1299 = '300°'
  3128 = '30°'
  3271 = '330°'
  1371 = '60°'
  2194 = '90°'
  920 = 'Awindup max'
  427 = 'Awindup min'
  433 = 'Board Stat'
  563 = 'Board Status'
  418 = 'Conv 0'
  84 = 'Conv 1'
  333 = 'Conv 10'
  797 = 'Conv 11'
  773 = 'Conv 12'
  174 = 'Conv 13'
  24 = 'Conv 14'
  818 = 'Conv 15'
  589 = 'Conv 2'
  856 = 'Conv 3'
  324 = 'Conv 4'
  432 = 'Conv 5'
  215 = 'Conv 6'
  172 = 'Conv 7'
  569 = 'Conv 8'
  394 = 'Conv 9'
  135 = 'Converters'
  253 = 'Converters gen'
  765 = 'Converters generation'
  565 = 'Energy_act'
  171 = 'Er_act_tot'
  966 = 'Er_reac_tot'
  521 = 'I ratio R'
  770 = 'I ratio S'
  867 = 'I ratio T'
  290 = 'Loads total'
  221 = 'Lost comms on / off'
  948 = 'Main'
  110 = 'Measures'
  227 = 'Meter\nconfig'
  539 = 'Meter cfg'
  741 = 'Meter config'
  792 = 'N mod'
  175 = 'N mode'
  610 = 'On/off'
  826 = 'Online'
  420 = 'P control Open Loop'
  224 = 'P control out'
  851 = 'P invert PI'
  887 = 'P loop'
  321 = 'P measured'
  206 = 'P net'
  64 = 'P PI invert'
  899 = 'P safety'
  264 = 'Phase P_min'
  228 = 'PI +Kp_min'
  875 = 'PI Kp'
  479 = 'PI Kp_min'
  257 = 'PI TI'
  43 = 'PoC net'
  392 = 'P_3ph'
  113 = 'P_control'
  992 = 'P_measured'
  312 = 'P_reference'
  538 = 'Q control Open Loop'
  961 = 'Q control out'
  61 = 'Q invert PI'
  836 = 'Q measured'
  625 = 'Q safety'
  220 = 'Q_3ph'
  276 = 'Q_control'
  346 = 'Q_reference'
  1101 = 'S minalç'
  229 = 'S nominal'
  161 = 'S nominalç'
  309 = 'Sat max'
  659 = 'Sat min'
  255 = 'SS-PPC ON/OFF'
  784 = 'V ratio RS'
  616 = 'V ratio ST'
  833 = 'V ratio TR'
  782 = 'V_line avg'
  530 = 'V_phase avg'
  472 = '_3ph'
END_TEXTLIST

// ---- VISUs/00_Main/Main.TcVIS
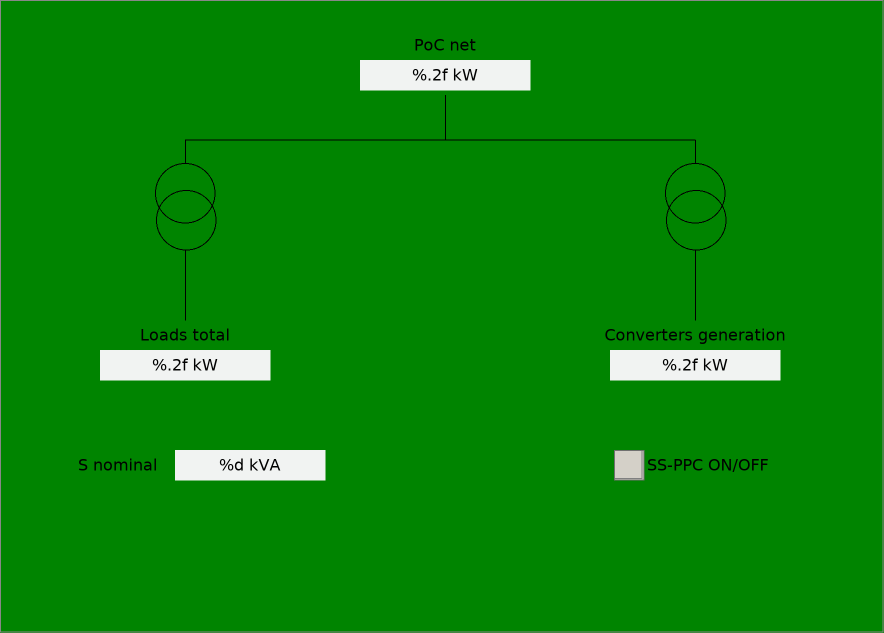
VISUALIZATION Main  // 884x633
    Rectangle (360,60 170x30), "%.2f kW", text variable: GVL_POWERMETER.M_board_P_kW
    Rectangle (390,30 110x30), "PoC net"
    Rectangle (610,350 170x30), "%.2f kW", text variable: GVL_POWERMETER.P_converters_tot
    Rectangle (605,320 180x30), "Converters generation"
    Rectangle (100,350 170x30), "%.2f kW", text variable: GVL_POWERMETER.M_board_P_kW + GVL_POWERMETER.P_converters_tot
    Rectangle (130,320 110x30), "Loads total"
    Line (445,95) (445,140)
    Line (695,250) (695,320)
    Line (185,250) (185,320)
    Ellipse (156,190 60x60)
    Ellipse (155,163 60x60)
    Ellipse (666,190 60x60)
    Ellipse (665,163 60x60)
    Line (695,140) (695,163)
    Line (185,140) (185,163)
    Line (695,140) (185,140)
    Rectangle (175,450 150x30), "%d kVA", text variable: GVL_PLANT_DEF.Plant_capacity_nom
        OnMouseClick: write the text variable via Default
    Rectangle (75,450 92x30), "S nominal"
    Rectangle (644,450 211x30), "SS-PPC ON/OFF"
    Button (614,450 30x30), colour toggle: GVL_GUI.Conv_n_mode_button[13]
        OnMouseClick: toggle GVL_GUI.Conv_n_mode_button[13]
        OnMouseClick: execute {
            IF GVL_CONV_COMMS.Night_Mode_Active[13] = 0 THEN
            	GVL_CONV_COMMS.Comms_Control_Word[13]:= GVL_CONV_COMMS.Comms_Control_Word[13] OR 16#0002;
            ELSE
            	GVL_CONV_COMMS.Comms_Control_Word[13]:= GVL_CONV_COMMS.Comms_Control_Word[13] AND 16#FFFD;
            END_IF
        }
END_VISUALIZATION

// ---- VISUs/00_Main/Main_GUI.TcVIS
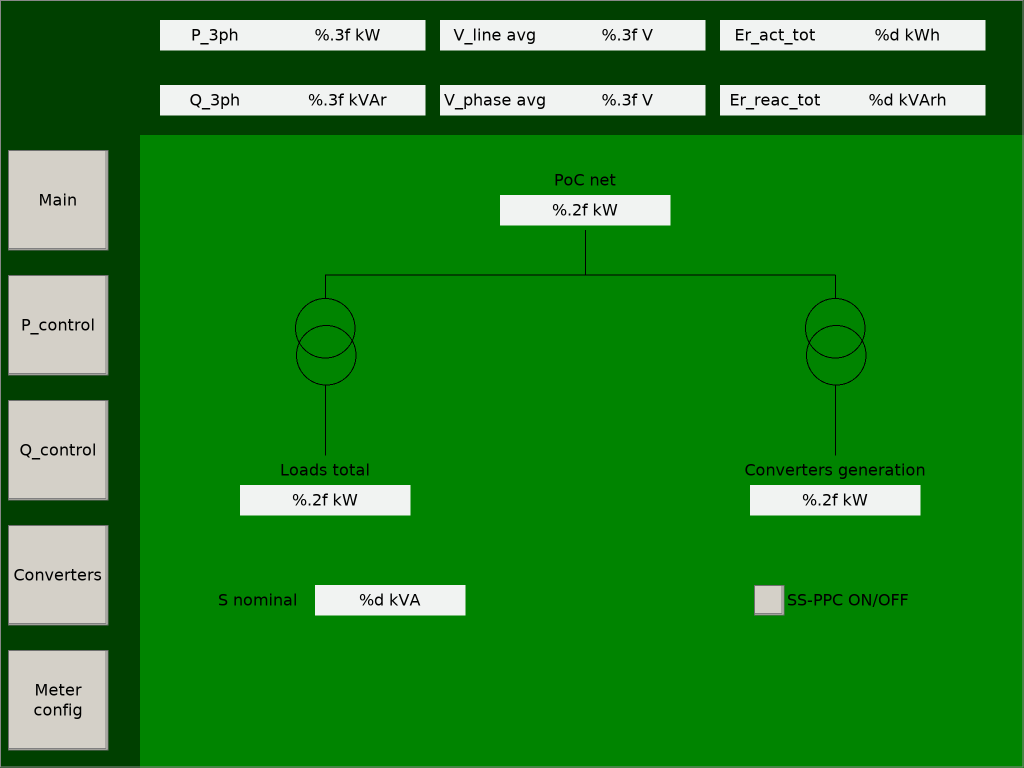
VISUALIZATION Main_GUI  // 1024x768
    Rectangle (160,20 110x30), "P_3ph"
    Rectangle (270,20 155x30), "%.3f kW", text variable: GVL_POWERMETER.Power_analyzer.P_kW
    Rectangle (160,85 110x30), "Q_3ph"
    Rectangle (270,85 155x30), "%.3f kVAr", text variable: GVL_POWERMETER.Power_analyzer.Q_kVAr
    Rectangle (440,20 110x30), "V_line avg"
    Rectangle (550,20 155x30), "%.3f V", text variable: GVL_POWERMETER.V_line_avg_Volt
    Rectangle (440,85 110x30), "V_phase avg"
    Rectangle (550,85 155x30), "%.3f V", text variable: GVL_POWERMETER.V_phase_avg_pu
    Rectangle (720,20 110x30), "Er_act_tot"
    Rectangle (830,20 155x30), "%d kWh", text variable: GVL_POWERMETER.Active_er_tot_kWh
    Rectangle (720,85 110x30), "Er_reac_tot"
    Rectangle (830,85 155x30), "%d kVArh", text variable: GVL_POWERMETER.React_er_tot_kVArh
    Button (8,150 100x100), "Main", colour toggle: GVL_GUI.main_button_logic
        OnMouseDown: execute {
            IF GVL_GUI.main_button_logic = 0 THEN
            	GVL_GUI.main_button_logic:= 1;
            	GVL_GUI.conv_button_logic:= 0;
            	GVL_GUI.pcontrol_button_logic:= 0;
            	GVL_GUI.qcontrol_button_logic:= 0;
            	GVL_GUI.meter_cfg_button_logic:= 0;
            	GVL_GUI.frame_indic:= 0;
            END_IF
        }
    Button (8,275 100x100), "P_control", colour toggle: GVL_GUI.pcontrol_button_logic
        OnMouseDown: execute {
            IF GVL_GUI.pcontrol_button_logic = 0 THEN
            	GVL_GUI.main_button_logic:= 0;
            	GVL_GUI.conv_button_logic:= 0;
            	GVL_GUI.pcontrol_button_logic:= 1;
            	GVL_GUI.qcontrol_button_logic:= 0;
            	GVL_GUI.meter_cfg_button_logic:= 0;
            	GVL_GUI.frame_indic:= 1;
            END_IF
        }
    Button (8,400 100x100), "Q_control", colour toggle: GVL_GUI.qcontrol_button_logic
        OnMouseDown: execute {
            IF GVL_GUI.qcontrol_button_logic = 0 THEN
            	GVL_GUI.main_button_logic:= 0;
            	GVL_GUI.conv_button_logic:= 0;
            	GVL_GUI.pcontrol_button_logic:= 0;
            	GVL_GUI.qcontrol_button_logic:= 1;
            	GVL_GUI.meter_cfg_button_logic:= 0;
            	GVL_GUI.frame_indic:= 2;
            END_IF
        }
    Button (8,525 100x100), "Converters", colour toggle: GVL_GUI.conv_button_logic
        OnMouseDown: execute {
            IF GVL_GUI.conv_button_logic = 0 THEN
            	GVL_GUI.main_button_logic:= 0;
            	GVL_GUI.conv_button_logic:= 1;
            	GVL_GUI.pcontrol_button_logic:= 0;
            	GVL_GUI.qcontrol_button_logic:= 0;
            	GVL_GUI.meter_cfg_button_logic:= 0;
            	GVL_GUI.frame_indic:= 3;
            END_IF
        }
    Button (8,650 100x100), "Meter config", colour toggle: GVL_GUI.meter_cfg_button_logic
        OnMouseDown: execute {
            IF GVL_GUI.meter_cfg_button_logic = 0 THEN
            	GVL_GUI.main_button_logic:= 0;
            	GVL_GUI.conv_button_logic:= 0;
            	GVL_GUI.pcontrol_button_logic:= 0;
            	GVL_GUI.qcontrol_button_logic:= 0;
            	GVL_GUI.meter_cfg_button_logic:= 1;
            	GVL_GUI.frame_indic:= 4;
            END_IF
        }
    Frame (140,135 884x633), frame switch variable: GVL_GUI.frame_indic
        shows Main()
        shows P_controller()
        shows Q_controller()
        shows Conv_handling()
        shows PM_config()
END_VISUALIZATION

// ---- VISUs/01_P_control/P_controller.TcVIS
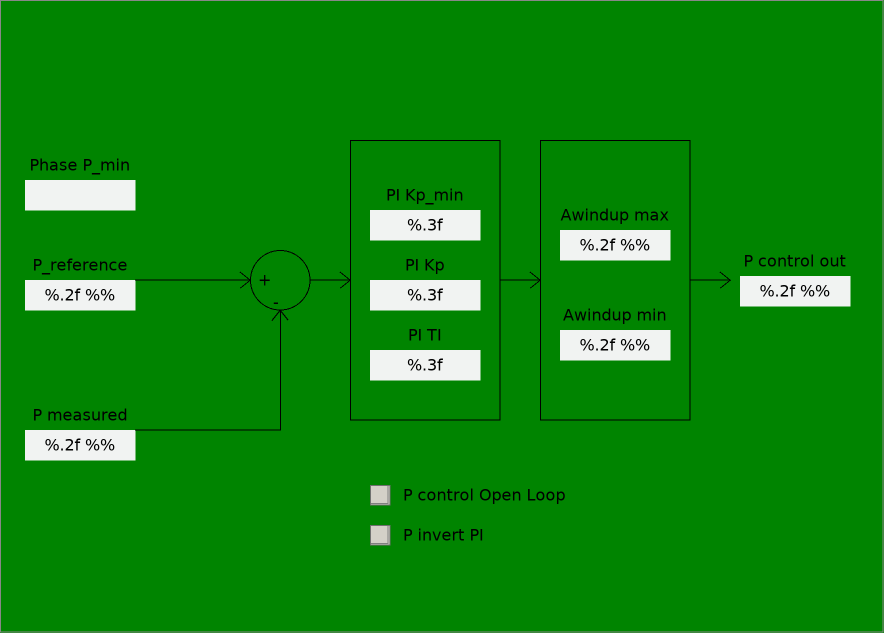
VISUALIZATION P_controller  // 884x633
    Rectangle (540,140 150x280)
    Rectangle (350,140 150x280)
    Rectangle (25,280 110x30), "%.2f %%", text variable: GVL_HANDLER.GUI_vars[P_reference]
        OnMouseDown: write the text variable via Default
    Rectangle (25,250 110x30), "P_reference"
    Rectangle (25,430 110x30), "%.2f %%", text variable: GVL_HANDLER.GUI_vars[P_feedback]
        OnMouseDown: write the text variable via Default
    Rectangle (25,400 110x30), "P measured"
    Line (250,280) (135,280)
    Ellipse (250,250 60x60)
    Line (280,430) (135,430)
    Line (280,310) (280,430)
    Line (288,320) (280,310)
    Line (272,320) (280,310)
    Line (250,280) (240,288)
    Line (250,280) (240,272)
    Line (350,280) (340,288)
    Line (350,280) (310,280)
    Line (350,280) (340,272)
    Rectangle (370,280 110x30), "%.3f", text variable: GVL_HANDLER.GUI_vars[P_kp]
        OnMouseClick: write the text variable via Default
    Rectangle (370,250 110x30), "PI Kp"
    Rectangle (370,350 110x30), "%.3f", text variable: GVL_HANDLER.GUI_vars[P_ti]
        OnMouseClick: write the text variable via Default
    Rectangle (370,320 110x30), "PI TI"
    Rectangle (370,210 110x30), "%.3f", text variable: GVL_HANDLER.GUI_vars[P_kp_min]
        OnMouseClick: write the text variable via Default
    Rectangle (370,180 110x30), "PI Kp_min"
    Line (540,280) (530,288)
    Line (540,280) (500,280)
    Line (540,280) (530,272)
    Rectangle (560,330 110x30), "%.2f %%", text variable: GVL_HANDLER.GUI_vars[P_low]
        OnMouseClick: write the text variable via Default
    Rectangle (560,300 110x30), "Awindup min"
    Rectangle (560,230 110x30), "%.2f %%", text variable: GVL_HANDLER.GUI_vars[P_high]
        OnMouseClick: write the text variable via Default
    Rectangle (560,200 110x30), "Awindup max"
    Line (730,280) (720,288)
    Line (730,280) (690,280)
    Line (730,280) (720,272)
    Rectangle (740,276 110x30), "%.2f %%", text variable: GVL_HANDLER.GUI_vars[P_output]
    Rectangle (740,246 110x30), "P control out"
    Rectangle (400,480 170x30), "P control Open Loop"
    Rectangle (400,520 170x30), "P invert PI"
    Button (370,485 20x20), colour toggle: GVL_GUI.P_OL_sel_button
        OnMouseClick: toggle GVL_HANDLER.GUI_vars[P_loop]
        OnMouseClick: execute {
            IF GVL_GUI.P_OL_sel_button = 0 THEN
            	GVL_GUI.P_OL_sel_button:= 1;
            ELSE
            	GVL_GUI.P_OL_sel_button:= 0;
            END_IF
        }
    Button (370,525 20x20), colour toggle: GVL_GUI.P_invert_button
        OnMouseClick: toggle GVL_HANDLER.GUI_vars[P_invert]
        OnMouseClick: execute {
            IF GVL_GUI.P_invert_button = 0 THEN
            	GVL_GUI.P_invert_button:= 1;
            ELSE
            	GVL_GUI.P_invert_button:= 0;
            END_IF
        }
    Rectangle (255,265 110x30), "+"
    Rectangle (270,287 110x30), "-"
    Rectangle (25,180 110x30), text list: 'P_min_indicator', text index: GVL_POWERMETER.P_min_indicator
    Rectangle (25,150 110x30), "Phase P_min"
END_VISUALIZATION

// ---- VISUs/01_P_control/P_min_indicator.TcTLO
TEXTLIST P_min_indicator
  0 = 'R'
  1 = 'S'
  2 = 'T'
   = ''
END_TEXTLIST

// ---- VISUs/02_Q_control/Q_controller.TcVIS
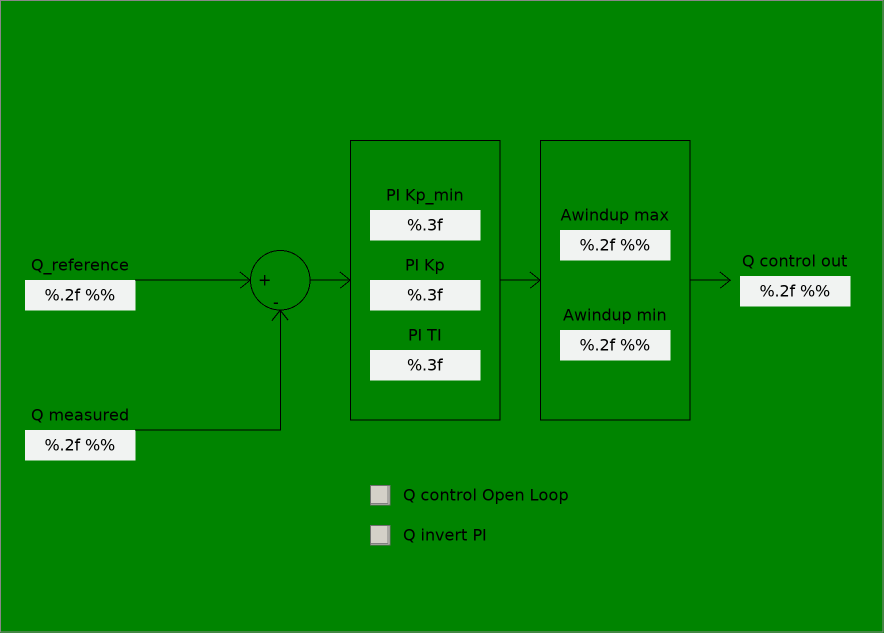
VISUALIZATION Q_controller  // 884x633
    Rectangle (540,140 150x280)
    Rectangle (350,140 150x280)
    Rectangle (25,280 110x30), "%.2f %%", text variable: GVL_HANDLER.GUI_vars[Q_reference]
        OnMouseDown: write the text variable via Default
    Rectangle (25,250 110x30), "Q_reference"
    Rectangle (25,430 110x30), "%.2f %%", text variable: GVL_HANDLER.GUI_vars[Q_feedback]
        OnMouseDown: write the text variable via Default
    Rectangle (25,400 110x30), "Q measured"
    Line (250,280) (135,280)
    Ellipse (250,250 60x60)
    Line (280,430) (135,430)
    Line (280,310) (280,430)
    Line (288,320) (280,310)
    Line (272,320) (280,310)
    Line (250,280) (240,288)
    Line (250,280) (240,272)
    Line (350,280) (340,288)
    Line (350,280) (310,280)
    Line (350,280) (340,272)
    Rectangle (370,280 110x30), "%.3f", text variable: GVL_HANDLER.GUI_vars[Q_kp]
        OnMouseClick: write the text variable via Default
    Rectangle (370,250 110x30), "PI Kp"
    Rectangle (370,350 110x30), "%.3f", text variable: GVL_HANDLER.GUI_vars[Q_ti]
        OnMouseClick: write the text variable via Default
    Rectangle (370,320 110x30), "PI TI"
    Rectangle (370,210 110x30), "%.3f", text variable: GVL_HANDLER.GUI_vars[Q_kp_min]
        OnMouseClick: write the text variable via Default
    Rectangle (370,180 110x30), "PI Kp_min"
    Line (540,280) (530,288)
    Line (540,280) (500,280)
    Line (540,280) (530,272)
    Rectangle (560,330 110x30), "%.2f %%", text variable: GVL_HANDLER.GUI_vars[Q_low]
        OnMouseClick: write the text variable via Default
    Rectangle (560,300 110x30), "Awindup min"
    Rectangle (560,230 110x30), "%.2f %%", text variable: GVL_HANDLER.GUI_vars[Q_high]
        OnMouseClick: write the text variable via Default
    Rectangle (560,200 110x30), "Awindup max"
    Line (730,280) (720,288)
    Line (730,280) (690,280)
    Line (730,280) (720,272)
    Rectangle (740,276 110x30), "%.2f %%", text variable: GVL_HANDLER.GUI_vars[Q_output]
    Rectangle (740,246 110x30), "Q control out"
    Rectangle (400,480 170x30), "Q control Open Loop"
    Rectangle (400,520 170x30), "Q invert PI"
    Button (370,485 20x20), colour toggle: GVL_GUI.Q_OL_sel_button
        OnMouseClick: toggle GVL_HANDLER.GUI_vars[Q_loop]
        OnMouseClick: execute {
            IF GVL_GUI.Q_OL_sel_button = 0 THEN
            	GVL_GUI.Q_OL_sel_button:= 1;
            ELSE
            	GVL_GUI.Q_OL_sel_button:= 0;
            END_IF
        }
    Button (370,525 20x20), colour toggle: GVL_GUI.Q_invert_button
        OnMouseClick: toggle GVL_HANDLER.GUI_vars[Q_invert]
        OnMouseClick: execute {
            IF GVL_GUI.Q_invert_button = 0 THEN
            	GVL_GUI.Q_invert_button:= 1;
            ELSE
            	GVL_GUI.Q_invert_button:= 0;
            END_IF
        }
    Rectangle (255,265 110x30), "+"
    Rectangle (270,287 110x30), "-"
END_VISUALIZATION

